    SEAL_FLATTENER_STATES.MovedFlattenersUpAndToClearance :                // Move flatteners to up state
                                                                    IF enable AND semiAutoModeSelected OR (autoModeSelected AND (_amMoveInToBagHolding OR _amMoveIn)) THEN
                                                                        state := SEAL_FLATTENER_STATES.MoveFlattenersIn;
                                                                        //ClearCommands();
                                                                    END_IF
                                        
                                                                    
    SEAL_FLATTENER_STATES.MoveFlattenersIn :                        // Move flatteners up and in
                                                                    //sealFlattenersHorizontalAxisMotor.NextSequence();    
                                                                    sealFlattenersHorizontalAxisMotor.MoveToPosition(position := inSetpoint, 
                                                                                                                        acceleration := horizontalAxisAccel,
                                                                                                                        deceleration := horizontalAxisDecel,
                                                                                                                        velocity := moveInSpeed);                                                    
                                                                    state := SEAL_FLATTENER_STATES.MovingFlattenersIn;
                                                                    
                                                                    
    SEAL_FLATTENER_STATES.MovingFlattenersIn :                        // If we did that command well move on 
                                                                        delay.IN := TRUE;
                                                                        IF delay.Q THEN
																			IF sealFlattenersHorizontalAxisMotor.CommandAcknowledged AND sealFlattenersHorizontalAxisMotor.InPosition THEN
																				state := SEAL_FLATTENER_STATES.MovedFlattenersIn;
                                                                           		delay.IN := FALSE;    
																			END_IF
                                                                        END_IF 
                                                                    
    SEAL_FLATTENER_STATES.MovedFlattenersIn :                        // Now that we're up and in move to down and 4 corners/bag holding
                                                                    IF enable AND semiAutoModeSelected OR (autoModeSelected AND _amMoveInToBagHolding) THEN
                                                                        state := SEAL_FLATTENER_STATES.MoveFlattenersDown;
                                                                        ClearCommands();
                                                                    END_IF    
    
    SEAL_FLATTENER_STATES.MoveFlattenersDown :            // Do moves for down and bag holding
                                                                        
                                                                        sealFlattenersVerticalAxis.Extend();
                                                                                                                                                                                
                                                                        state := SEAL_FLATTENER_STATES.MovingFlattenersDown;
                                                                        
    SEAL_FLATTENER_STATES.MovingFlattenersDown :            
                                                                        //IF sealFlattenersVerticalAxis.CommandAcknowledged AND sealFlattenersVerticalAxis.InPosition THEN
                                                                       	fingersDownDelay.IN := TRUE;
																	  	IF fingersDownDelay.Q THEN
																			state := SEAL_FLATTENER_STATES.MovedFlattenersDown;
																			fingersDownDelay.IN := FALSE;
																		END_IF 
																		
                                                                        //END_IF 
                                                                        
    SEAL_FLATTENER_STATES.MovedFlattenersDown :            state := SEAL_FLATTENER_STATES.MoveFlattenersToBagHolding;
                                                                    
                                                                    
    SEAL_FLATTENER_STATES.MoveFlattenersToBagHolding :            // Do moves for down and bag holding
                                                                        //sealFlattenersHorizontalAxisMotor.NextSequence();    
                                                                        sealFlattenersHorizontalAxisMotor.MoveToPositionTorque(position := bagHoldingSetpoint, 
                                                                                                                        acceleration := horizontalAxisAccel,
                                                                                                                        deceleration := horizontalAxisDecel,
                                                                                                                        velocity := moveBagHoldingSpeed,
																														current := bagHoldingCurrentMSF);                                                
                                                                        state := SEAL_FLATTENER_STATES.MovingFlattenersToBagHolding;
                                                                        
    SEAL_FLATTENER_STATES.MovingFlattenersToBagHolding :            delay.IN := TRUE;
                                                                        IF delay.Q THEN
																			IF sealFlattenersHorizontalAxisMotor.CommandAcknowledged THEN
																				state := SEAL_FLATTENER_STATES.MovedFlattenersToBagHolding;
                                                                            	delay.IN := FALSE; 
																			END_IF   
                                                                        END_IF 
                                                                        
    SEAL_FLATTENER_STATES.MovedFlattenersToBagHolding :            state := SEAL_FLATTENER_STATES.Idle;
																		HMIData.motorizedSealFlattenerCycles.Increment();
                                                                        Globals.motorizedSealFlattenersCount := Globals.motorizedSealFlattenersCount +1;
                                                                        Globals.sealFlattenerFingersCount := Globals.sealFlattenerFingersCount +1;
    SEAL_FLATTENER_STATES.Ready :
    SEAL_FLATTENER_STATES.Fault :
END_CASE

METHOD PRIVATE ClearCommands
VAR_INPUT
END_VAR
// Clear all commands from auto mode
_amMoveOut := FALSE;
_amMoveClearance := FALSE;
_amMoveInToBagHolding := FALSE;
_amMoveIn := FALSE;
END_METHOD

METHOD AutoMoveOut
VAR_INPUT
END_VAR
_amMoveOut := TRUE;
END_METHOD

PROPERTY Mode : DEVICE_MODES
SET
_mode := Mode;
END_SET
GET
Mode := _mode;
END_GET
END_PROPERTY

PROPERTY Ready : BOOL
GET
Ready := _ready;
END_GET
SET
_ready := Ready;
END_SET
END_PROPERTY

METHOD AutoMoveToClearance
VAR_INPUT
END_VAR
_amMoveClearance := TRUE;
END_METHOD

METHOD AutoMoveToBagHolding
VAR_INPUT
END_VAR
_amMoveInToBagHolding := TRUE;
END_METHOD

METHOD AutoMoveIn : BOOL
VAR_INPUT
END_VAR
_amMoveIn := TRUE;
END_METHOD

END_FUNCTION_BLOCK

// Device/Application/FBs/Cylinders/ICylinder
INTERFACE ICylinder

METHOD Extend
VAR_INPUT
END_VAR
END_METHOD

METHOD Execute
VAR_INPUT
END_VAR
END_METHOD

METHOD Retract
VAR_INPUT
END_VAR
END_METHOD

END_INTERFACE

// Device/Application/FBs/Motors/Festo/FB_FestoMotor
FUNCTION_BLOCK FB_FestoMotor IMPLEMENTS IPositionableMotor, IStoredProgramMotor
VAR_INPUT
    deviceType : FML.E_FML_DEVICE_TYPE;                            //Must define drive type
    isFPCActive : BOOL;    
    ptrReadFHPPRegister : POINTER TO WORD;
    ptrReadFPCRegister : POINTER TO WORD;
    ptrWriteFHPPRegister : POINTER TO WORD;
    ptrWriteFPCRegister : POINTER TO WORD;                                        //Toggle if FPC(Festo Parameter Chanel) is active or not
END_VAR
VAR_IN_OUT
    //modbusReadRegisters :  ARRAY[0..7] OF WORD;        //Inputs from drive
    //modbusWriteRegisters : ARRAY[0..7] OF WORD;    //Outputs to write to drive

END_VAR
VAR_OUTPUT
END_VAR
VAR
    //Required datatypes for the Festo motor blocks
    FHPP_IN     :ARRAY[0..7] OF BYTE;
    FHPP_OUT     :ARRAY[0..7] OF BYTE;
    FPC_IN         :ARRAY[0..7] OF BYTE;
    FPC_OUT     :ARRAY[0..7] OF BYTE;
    ReadAxis            :FML.FML_Read;
    DATA_REF_Axis         :FML.DT_FML_REF;
    CRTL_Axis            :FML.FHPP_CTRL;
    PNU_Axis            :FML.FPC_PNU;
    MULTI_Axis            :FML.FPC_MULTI;    
    DIRMP_Axis            :FML.FPC_DIRMP;
    DIAG_Axis            :FML.FPC_DIAG;
    DIAG_BUFF_Axis        :FML.FPC_DIAG_BUFFER;
    DATA_OBJECT_Axis    :FML.FPC_DATA_OBJECT;
    FILE_Axis            :FML.FPC_FILE;
    FILE_ARRAY_Axis        :FML.FPC_FILE_ARRAY;
    WriteAxis            :FML.FML_Write;

    //Regular variables
    ptrModbusMemory : POINTER TO ARRAY[0..7] OF BYTE; 
    commandSuccessful : BOOL;    //Modbus Command was successful
    homeRequiredIndication : BOOL; //Home required indication
    homingActive : BOOL;            //Homing active
    removeStartCommandTimer : Standard.TON := (PT := T#100MS);
    startAckONS : Standard.R_TRIG;
    _sendStart : BOOL;
END_VAR
VAR_STAT    
    //Make these static to share amongst all instances of the Festo motors
    ARY_DATA_FILE        :ARRAY[0..25000] OF BYTE;
    MultiParam             :ARRAY [0..7] OF DT_FML_PRM_DESCRIPTION :=[
                                            (PNU:=404, SUBINDEX:=1, ACCESS:=0, VALUE:=0, LENGTH:=0),
                                            (PNU:=404, SUBINDEX:=1, ACCESS:=1, VALUE:=100, LENGTH:=4),
                                            (PNU:=404, SUBINDEX:=1, ACCESS:=0, VALUE:=0, LENGTH:=0),
                                            (PNU:=404, SUBINDEX:=2, ACCESS:=0, VALUE:=0, LENGTH:=0),
                                            (PNU:=404, SUBINDEX:=2, ACCESS:=1, VALUE:=200, LENGTH:=4),
                                            (PNU:=404, SUBINDEX:=2, ACCESS:=0, VALUE:=0, LENGTH:=0),
                                            (PNU:=404, SUBINDEX:=1, ACCESS:=1, VALUE:=111, LENGTH:=4),
                                            (PNU:=404, SUBINDEX:=1, ACCESS:=0, VALUE:=0, LENGTH:=0)];
                                            
END_VAR

METHOD ExecuteStoredProgram
VAR_INPUT
    (*Program number to execute*)
    programNumber    : INT;
END_VAR
InitDrive();
IF InPosition AND CRTL_Axis.ActualRecordNo = programNumber THEN
    commandSuccessful := TRUE;
ELSE
    CRTL_Axis.RecordNo := programNumber;
    _sendStart := TRUE;
END_IF
END_METHOD

PROPERTY Homing : BOOL
GET
Homing := homingActive;
END_GET
END_PROPERTY

PROPERTY HomeRequired : BOOL
GET
HomeRequired := homeRequiredIndication;
END_GET
SET
homeRequiredIndication := HomeRequired;
END_SET
END_PROPERTY

{attribute 'monitoring' := 'variable'}
PROPERTY CurrentPosition : REAL
GET
{warning: 'TODO: Find out actual conversion factor'}    
CurrentPosition := (DINT_TO_REAL(CRTL_Axis.ActualPosition)/100);
END_GET
END_PROPERTY

METHOD Execute
VAR_INPUT
END_VAR


//Check to make sure we have a valid reference.  Disable complier warning since we're doing the check
//{warning disable C0371}
(*
IF NOT __ISVALIDREF(ptrReadFHPPRegister) 
    OR NOT __ISVALIDREF(ptrReadFPCRegister) 
    OR NOT __ISVALIDREF(ptrWriteFHPPRegister)
    OR NOT __ISVALIDREF(ptrWriteFPCRegister)
THEN
     RETURN;
END_IF
*)



//Convert array of bytes to array of words. Playin' with pointers!
ptrModbusMemory := ptrReadFHPPRegister;
FHPP_IN := ptrModbusMemory^; 
ptrModbusMemory := ptrReadFPCRegister;
FPC_IN := ptrModbusMemory^;
ptrModbusMemory := ptrWriteFHPPRegister;
ptrModbusMemory^ := FHPP_OUT; 
ptrModbusMemory := ptrWriteFPCRegister;
ptrModbusMemory^ := FPC_OUT;

// Function block calls for axis
ReadAxis(
    FML_REF            := DATA_REF_Axis,
    Modbus            := FALSE,
    HighByteFirst    := TRUE,
    DeviceType        := deviceType,
    FPC_active        := isFPCActive,
    
    FHPP_Source        := FHPP_IN,
    FPC_Source        := FPC_IN);    
CRTL_Axis(
    FML_REF            := DATA_REF_Axis);    
PNU_Axis(
    FML_REF            := DATA_REF_Axis);
MULTI_Axis(
    FML_REF            := DATA_REF_Axis,
    SizeOfParam        := SIZEOF(MultiParam),
    AdrOfParam        := ADR(MultiParam));
DIRMP_Axis(
    FML_REF            := DATA_REF_Axis);    
DIAG_Axis(
    FML_REF            := DATA_REF_Axis);
DIAG_BUFF_Axis(
    FML_REF            := DATA_REF_Axis);
DATA_OBJECT_Axis(
    FML_REF            := DATA_REF_Axis);
FILE_Axis(
    FML_REF            := DATA_REF_Axis);
FILE_ARRAY_Axis(
    FML_REF            := DATA_REF_Axis,
    SizeOfFileArray    := SIZEOF(ARY_DATA_FILE),
    AdrOfFileArray    := ADR(ARY_DATA_FILE));    
WriteAxis(
    FML_REF            := DATA_REF_Axis,
    FHPP_Target        => FHPP_OUT,
    FPC_Target        => FPC_OUT);
{warning 'TODO: Remove this hack to clear start command if error occurs'}
removeStartCommandTimer(IN := CRTL_Axis.StartTask OR CRTL_Axis.AckStart);
//removeStartCommandTimer(IN := CRTL_Axis.AckStart);
startAckONS(CLK := CRTL_Axis.AckStart);    
//IF removeStartCommandTimer.Q THEN
IF _sendStart AND NOT CRTL_Axis.AckStart THEN
    CRTL_Axis.StartTask := TRUE;
    _sendStart := FALSE;
END_IF

IF startAckONS.Q OR removeStartCommandTimer.Q THEN
    CRTL_Axis.StartTask := FALSE;
    commandSuccessful := TRUE;
END_IF
//Set Home required indication
homeRequiredIndication S= NOT CRTL_Axis.HomingValid;
//commandSuccessful S= CRTL_Axis.AckStart;
//{warning restore C0371}
END_METHOD

{attribute 'monitoring' := 'variable'}
PROPERTY CommandAcknowledged : BOOL
GET
CommandAcknowledged := commandSuccessful;
END_GET
END_PROPERTY

METHOD Stop
commandSuccessful := FALSE;
CRTL_Axis.EnableDrive := TRUE;
CRTL_Axis.Halt := TRUE;
CRTL_Axis.Stop := FALSE;
END_METHOD

{attribute 'monitoring' := 'variable'}
PROPERTY ActiveStoredProgramNumber : INT
GET
ActiveStoredProgramNumber := CRTL_Axis.ActualRecordNo;
END_GET
END_PROPERTY

METHOD PRIVATE InitDrive
VAR_INPUT
END_VAR
//Initialize the drive to prepare for a move
CRTL_Axis.EnableDrive := TRUE;
CRTL_Axis.Halt := TRUE;
CRTL_Axis.Stop := TRUE;    
//CRTL_Axis.StartTask := FALSE;
commandSuccessful := FALSE;
END_METHOD

PROPERTY Moving : BOOL
GET
Moving := CRTL_Axis.DriveIsMoving;
END_GET
END_PROPERTY

{warning 'add method implementation '}
METHOD MoveDistance
VAR_INPUT
    (*Distance to move in inches*)
    distance    : REAL;
    (*Acceleration in RPM/sec*)
    acceleration    : INT;
    (*Deceleration in RPM/sec*)
    deceleration    : INT;
    (*Velocity in .25RPM*)
    velocity    : INT;
END_VAR
END_METHOD

{attribute 'monitoring' := 'variable'}
PROPERTY InPosition : BOOL
GET
InPosition := CRTL_Axis.MC;
END_GET
END_PROPERTY

{warning 'add method implementation '}
METHOD MoveToPosition
VAR_INPUT
    (*Position to move to in inches*)
    position    : REAL;
    (*Acceleration in RPM/sec*)
    acceleration    : INT;
    (*Deceleration in RPM/sec*)
    deceleration    : INT;
    (*Velocity in .25RPM*)
    velocity    : INT;
END_VAR
END_METHOD

METHOD HomeNow
CRTL_Axis.StartHoming := TRUE;
END_METHOD

END_FUNCTION_BLOCK

// Device/Application/FBs/Motors/IPositionableMotor
INTERFACE IPositionableMotor

PROPERTY Homing : BOOL
GET
END_GET
END_PROPERTY

PROPERTY Moving : BOOL        //Motor is Moving
GET
END_GET
END_PROPERTY

PROPERTY InPosition : BOOL        //Motor is in position
GET
END_GET
END_PROPERTY

PROPERTY CurrentPosition : REAL        //Current motor position in Inches
GET
END_GET
END_PROPERTY

METHOD Stop
VAR_INPUT
END_VAR
END_METHOD

PROPERTY CommandAcknowledged : BOOL        //Command acked from drive
GET
END_GET
END_PROPERTY

METHOD HomeNow
VAR_INPUT
END_VAR
END_METHOD

METHOD MoveToPosition
VAR_INPUT
    position : REAL;        //Position to move to in inches
    acceleration : INT;        //Acceleration in RPM/sec
    deceleration : INT;        //Deceleration in RPM/sec
    velocity : INT;            //Velocity in .25RPM
END_VAR
END_METHOD

PROPERTY HomeRequired : BOOL
GET
END_GET
SET
END_SET
END_PROPERTY

METHOD MoveDistance
VAR_INPUT
    distance : REAL;        //Distance to move in inches
    acceleration : INT;        //Acceleration in RPM/sec
    deceleration : INT;        //Deceleration in RPM/sec
    velocity : INT;            //Velocity in .25RPM
END_VAR
END_METHOD

END_INTERFACE

// Device/Application/FBs/Motors/IStoredProgramMotor
INTERFACE IStoredProgramMotor

PROPERTY ActiveStoredProgramNumber : INT
GET
END_GET
END_PROPERTY

METHOD ExecuteStoredProgram
VAR_INPUT
    programNumber : INT;        //Program number to execute
END_VAR
END_METHOD

END_INTERFACE

// Device/Application/FBs/Fault/FB_ONS
FUNCTION_BLOCK FB_ONS
VAR_INPUT
	CLK : BOOL;
END_VAR
VAR_OUTPUT
	OSR : BOOL;
	OSF : BOOL;
END_VAR
VAR
	CLK_OSR : R_TRIG;
	CLK_OSF : F_TRIG;
END_VAR

CLK_OSR(CLK := CLK, Q=> OSR);
CLK_OSF(CLK := CLK, Q=> OSF);

END_FUNCTION_BLOCK

// Device/Application/FBs/Motors/Applied Motion/FB_AppliedMotionStepServoEIPBaseQX
FUNCTION_BLOCK FB_AppliedMotionStepServoEIPBaseQX IMPLEMENTS IPositionableMotor, IStoredProgramMotor
VAR_INPUT
    ptrEIPInputs : POINTER TO ARRAY[0..13] OF  DINT;
    ptrEIPOutputs : POINTER TO ARRAY[0..15] OF DINT;
    faultHandler : REFERENCE TO FB_FaultHandler;
	commFail : BOOL;
    stepsPerInchSetpoint : INT;             //Steps per inch setpoint
    reversePolarity : BOOL;                 //0 = Normal, 1 = reversed polarity for display
    jogAccelSetpoint : INT;        //Point-to-Point Acceleration (AC) Setpoint
    jogDecelSetpoint : INT;        //Point-to-Point Deceleration (DE) Setpoint
    jogVelocitySetpoint : INT;                //Velocity (VE) Setpoint
    pointToPointAccelSetpoint : INT;        //Point-to-Point Acceleration (AC) Setpoint
    pointToPointDecelSetpoint : INT;        //Point-to-Point Deceleration (DE) Setpoint
    velocitySetpoint : INT;                //Velocity (VE) Setpoint
	defaultCurrentSetpoint : DINT;
	sclCommand : DINT;						// SCL Command from 
	parameter1 : DINT;						// Data/SCL parameter 1
	parameter2 : DINT;						// Data/SCL parameter 2
    distanceSetpointInches : REAL;        //Distance setpoint in inches Setpoint
    moveDistanceManualPB : BOOL;            //Move distance pushbutton
    movePositionManualPB : BOOL;            //Move position pushbutton
	isHomable : BOOL;
END_VAR
VAR_IN_OUT
    //slave : IoDrvModbusTCP.ModbusTCPSlave;                    //Slave ModbusTCP Object
END_VAR
VAR
    absolutePositionSteps : DINT; //Immediate Absolute Position in steps
    distanceToMoveInSteps : DINT;        //Distance Setpoint to Drive
    stepServoStatusRaw : INT; //Raw step servo status over modbus
	stepServoAlarmCodeRaw : INT; // Ras Step Servo alarm code word
	currentLimit : DINT;
    commands : FB_StepServoCommands();
    commandSuccessful : BOOL;    //Modbus Command was successful
    commandSuccessfulONS : R_TRIG;    //Modbus Command was successful
    commandSentONS : R_TRIG;    //Modbus Command was successful
    homeRequiredIndication : BOOL; //Home required indication.
    driveInputs : ARRAY[0..13] OF DINT;        // Inputs from drive over EIP
    driveOutputs : ARRAY[0..15] OF DINT;    // Outputs to drive over EIP
    interfaceToPass : IFault;
    faultListRegisterSuccess : BOOL;        // Registering in fault list successful
    _faulted : BOOL;                    // Motor Faulted
	_reset : BOOL;			//Reset Motor
	_homeNow : BOOL;
	homingOSF : F_TRIG;
	
	IECReferenceGood : BOOL;
END_VAR
VAR_OUTPUT
    absolutePositonInches : REAL; //Immediate Absolute Positon in inches
    velocity : INT;    //Velocity (VE) Input from Drive
    status : StepServoStatusFB; //Status of servo
	alarms : FB_StepServoAlarms; // Alarms from Drive
    QSegmentRunning : INT; //Current Q program running from Drive
	faults : StepServoFaultsType;
END_VAR


IF NOT faultListRegisterSuccess THEN
    faultListRegisterSuccess := RegisterWithFaultHandler();
END_IF

METHOD Execute
VAR_INPUT
END_VAR
//    Function Block: AppliedMotionStepServo
//    Description: This block provides an abstraction for a Ethernet I/P Applied Motion Step Servo
//    Created by: Ben Hess
//    Created Date: May 11th, 2018

// Use pointers for EIP memory register locations
driveInputs := ptrEIPInputs^;

ptrEIPOutputs^ := driveOutputs;
alarms(alarmCode := stepServoAlarmCodeRaw, faults := faults);

IF currentLimit = 0 THEN 
	currentLimit := defaultCurrentSetpoint;
END_IF
//Map raw EIP Registers to parameters
absolutePositionSteps := driveInputs[6];
velocity := DINT_TO_INT(driveInputs[8]);
stepServoStatusRaw := DINT_TO_INT(driveInputs[0]);

driveOutputs[4] := velocitySetpoint;
driveOutputs[5] := pointToPointAccelSetpoint;
driveOutputs[6] := pointToPointDecelSetpoint;
driveOutputs[7] := distanceToMoveInSteps;
driveOutputs[8] := currentLimit;
driveOutputs[9] := sclCommand;
driveOutputs[10] := parameter1;
driveOutputs[11] := parameter2;
driveOutputs[12] := currentLimit;
driveOutputs[13] := currentLimit + 1;
driveOutputs[0] := commands.commandWord;
// Step servo command bits handler
commands();
//Convert Distance setpoint to steps.  Reverse polarity for display purposes if needed. 

absolutePositonInches := (DINT_TO_REAL(absolutePositionSteps) / INT_TO_REAL(stepsPerInchSetpoint));

//Homing required from motor - for now just if there was an initialization seen.
homeRequiredIndication S= status.initializing OR Globals.firstScan OR _faulted OR driveInputs[11].0;

homingOSF(CLK := status.homing);
IF NOT driveInputs[11].0 THEN
	homeRequiredIndication := FALSE;
END_IF

commandSentONS(CLK := commands.commandSent);

IF commandSentONS.Q THEN
	commandSuccessful := TRUE;
END_IF

commandSuccessfulONS(CLK := commandSuccessful);
IF commandSuccessfulONS.Q THEN
	//parameter1 := 0;
	//velocitySetpoint := 0;
	//pointToPointAccelSetpoint := 0;
	//pointToPointDecelSetpoint := 0;
	//distanceToMoveInSteps := 0;
END_IF


IF _reset AND (status.driveFaulted OR status.alarmPresent) THEN
	commands.alarmReset := TRUE;
	_reset := FALSE;
END_IF

IF reversePolarity THEN
    absolutePositonInches := absolutePositonInches * -1; 
END_IF

//Get Servo Status and unpack
status(statusCode := StepServoStatusRaw);

//Bit-packing for LONG types over Modbus

_faulted := status.driveFaulted OR status.alarmPresent OR commFail;

//Manual moves for motor
IF moveDistanceManualPB THEN
    MoveDistance(distance := distanceSetpointInches, acceleration := pointToPointAccelSetpoint, deceleration := pointToPointDecelSetpoint, velocity := velocitySetpoint);
    moveDistanceManualPB := FALSE;
END_IF

IF movePositionManualPB THEN
    MoveToPosition(position := distanceSetpointInches, acceleration := pointToPointAccelSetpoint, deceleration := pointToPointDecelSetpoint, velocity := velocitySetpoint);
    movePositionManualPB := FALSE;
END_IF


faults.commFail.faultTrigger := commFail AND Globals.machinePowerOK;
faults.notHomed.faultTrigger := homeRequiredIndication AND isHomable;
END_METHOD

{attribute 'monitoring' := 'variable'}
PROPERTY CommandAcknowledged : BOOL
GET
CommandAcknowledged := commandSuccessful;
END_GET
END_PROPERTY

METHOD HomeNow
commandSuccessful := FALSE;
parameter1 := 1;
pointToPointAccelSetpoint := 1000;
pointToPointDecelSetpoint := 1000;
velocitySetpoint := 2500;
distanceToMoveInSteps := 0;
commands.sendQAndExecute := TRUE;

//homeRequiredIndication := FALSE;
END_METHOD

{attribute 'monitoring' := 'variable'}
PROPERTY HomeRequired : BOOL
SET
homeRequiredIndication := HomeRequired;
END_SET
GET
HomeRequired := homeRequiredIndication;
END_GET
END_PROPERTY

{attribute 'monitoring' := 'variable'}
PROPERTY Moving : BOOL
GET
Moving := status.moving;
END_GET
END_PROPERTY

{attribute 'monitoring' := 'variable'}
PROPERTY ActiveStoredProgramNumber : INT
GET
ActiveStoredProgramNumber := QSegmentRunning;
END_GET
END_PROPERTY

{attribute 'monitoring' := 'variable'}
PROPERTY InPosition : BOOL
GET
InPosition := status.inPosition;
END_GET
END_PROPERTY

METHOD MoveDistanceTorque
VAR_INPUT
	(*Distance to move in inches*)
    distance    : REAL;
    (*Acceleration in RPM/sec*)
    acceleration    : INT;
    (*Deceleration in RPM/sec*)
    deceleration    : INT;
    (*Velocity in .25RPM*)
    velocity    : INT;
	(*Current in .01A*)
	current : DINT;
END_VAR
//This method preps the data to send to the drive and triggers the send.
//Set distance and unpack to prep data to send to motor

commandSuccessful := FALSE;

distanceToMoveInSteps := REAL_TO_DINT((distance) * stepsPerInchSetpoint);
IF reversePolarity THEN
    distanceToMoveInSteps := distanceToMoveInSteps * -1;
END_IF

pointToPointAccelSetpoint := acceleration;
pointToPointDecelSetpoint := deceleration;
velocitySetpoint := velocity;
currentLimit := current;

parameter1 := 2;
commands.SendQAndExecute := TRUE;
END_METHOD

(* This will be called if the machine is faulted*)
METHOD MachineFaulted
END_METHOD

{attribute 'monitoring' := 'variable'}
PROPERTY Faulted : BOOL
GET
Faulted := _faulted;
END_GET
SET
END_SET
END_PROPERTY

METHOD MoveToPosition
VAR_INPUT
    (*Position to move to in inches*)
    position    : REAL;
    (*Acceleration in RPM/sec*)
    acceleration    : INT;
    (*Deceleration in RPM/sec*)
    deceleration    : INT;
    (*Velocity in .25RPM*)
    velocity    : INT;
END_VAR
commandSuccessful := FALSE;

distanceToMoveInSteps := REAL_TO_DINT((position) * stepsPerInchSetpoint);
IF reversePolarity THEN
    distanceToMoveInSteps := distanceToMoveInSteps * -1;    
END_IF

pointToPointAccelSetpoint := acceleration;
pointToPointDecelSetpoint := deceleration;
velocitySetpoint := velocity;
currentLimit := defaultCurrentSetpoint;

commands.feedToPosition := TRUE;
END_METHOD

METHOD MoveToPositionTorque
VAR_INPUT
	(*Position to move to in inches*)
    position    : REAL;
    (*Acceleration in RPM/sec*)
    acceleration    : INT;
    (*Deceleration in RPM/sec*)
    deceleration    : INT;
    (*Velocity in .25RPM*)
    velocity    : INT;
	(*Current in .01A*)
	current : DINT;
END_VAR
commandSuccessful := FALSE;

distanceToMoveInSteps := REAL_TO_DINT((position) * stepsPerInchSetpoint);
IF reversePolarity THEN
    distanceToMoveInSteps := distanceToMoveInSteps * -1;    
END_IF

pointToPointAccelSetpoint := acceleration;
pointToPointDecelSetpoint := deceleration;
velocitySetpoint := velocity;
currentLimit := current;

commands.feedToPosition := TRUE;
THIS^.Execute();
END_METHOD

//{warning 'add method implementation '}
METHOD Stop
commandSuccessful := FALSE;
commands.StopNormal := TRUE;
END_METHOD

METHOD MoveDistance
VAR_INPUT
    (*Distance to move in inches*)
    distance    : REAL;
    (*Acceleration in RPM/sec*)
    acceleration    : INT;
    (*Deceleration in RPM/sec*)
    deceleration    : INT;
    (*Velocity in .25RPM*)
    velocity    : INT;
END_VAR
//This method preps the data to send to the drive and triggers the send.
//Set distance and unpack to prep data to send to motor

commandSuccessful := FALSE;

distanceToMoveInSteps := REAL_TO_DINT((distance) * stepsPerInchSetpoint);
IF reversePolarity THEN
    distanceToMoveInSteps := distanceToMoveInSteps * -1;
END_IF

pointToPointAccelSetpoint := acceleration;
pointToPointDecelSetpoint := deceleration;
velocitySetpoint := velocity;
currentLimit := defaultCurrentSetpoint;

commands.feedToLength := TRUE;
END_METHOD

{attribute 'monitoring' := 'variable'}
PROPERTY CurrentPosition : REAL  //Current motor position in Inches
GET
CurrentPosition := absolutePositonInches;
END_GET
END_PROPERTY

{attribute 'monitoring' := 'variable'}
PROPERTY Homing : BOOL
GET
Homing := status.homing;
END_GET
END_PROPERTY

METHOD Reset : BOOL
VAR_INPUT
END_VAR
IF Faulted THEN
	_reset := TRUE;
	commands.AlarmReset := TRUE;
END_IF
commands.Enable := TRUE;
END_METHOD

METHOD RegisterWithFaultHandler : BOOL
// If faulthandler hasn't been initialized yet then do nothing.

(*
IF NOT __ISVALIDREF(faultHandler) THEN
     RETURN;
END_IF

interfaceToPass := THIS^;
faultHandler.registerFaultSource(interfaceToPass);
RegisterWithFaultHandler := TRUE;
*)
END_METHOD

METHOD ExecuteStoredProgram
VAR_INPUT
    (*Program number to execute*)
    programNumber    : INT;
END_VAR
parameter1 := programNumber;
commands.SendQAndExecute := TRUE;
END_METHOD

END_FUNCTION_BLOCK

// Device/Application/FBs/FB_FaultHandler
FUNCTION_BLOCK FB_FaultHandler
VAR_INPUT
END_VAR
VAR_OUTPUT
END_VAR
VAR
    faultSourceList : ARRAY[0..100] OF IFault;
    sourcesInList : INT;
END_VAR

METHOD registerFaultSource
VAR_INPUT
     faultSource : REFERENCE TO IFault;
END_VAR
faultSourceList[sourcesInList]:= faultSource;
sourcesInList:= sourcesInList + 1;
END_METHOD

END_FUNCTION_BLOCK

// Device/Application/ObjectHandling/IFault
INTERFACE IFault EXTENDS IAllObjects

METHOD Trigger
VAR_INPUT
END_VAR
END_METHOD

METHOD Ack
VAR_INPUT
END_VAR
END_METHOD

END_INTERFACE

// Device/Application/ObjectHandling/IAllObjects
INTERFACE IAllObjects EXTENDS __System.IQueryInterface

PROPERTY InstanceName : STRING
GET
END_GET
END_PROPERTY

END_INTERFACE

// Device/Application/FBs/Motors/Applied Motion/DataHandlers/FB_StepServoCommands
{analysis -166, -35, -36, -38, -148}
FUNCTION_BLOCK FB_StepServoCommands
VAR_INPUT
       
END_VAR
VAR_OUTPUT
    commandWord : DINT;
	commandSent : BOOL;
END_VAR
VAR
	_idleState : BOOL; // Idle State (Send this between repeated commands)
    _enable : BOOL; // Enable
    _disable : BOOL; // Disable
    _feedToLength : BOOL; // Start Move - FL
    _feedToPosition : BOOL; // Start Move - FP
    _feedToSensor : BOOL; // Start Move - FS (sensor)
    _feedToDoubleSensor : BOOL; // Start Move - FD (double sensor)
    _feedToSensorSafety : BOOL; // Start Move - FY (sensor w/ safety distance)
    _feedToSensorMask : BOOL; // Start Move - FM (sensor w/ mask distance)
    _feedAndSetOutput : BOOL; // Start Move - FO (set output)
    _feedSpeedChange : BOOL; // Start Move - FC
    _seekHome : BOOL; // Start Move - SH
    _findHome : BOOL; // Start Move - FH
    _followEncoder : BOOL; // Start Move - FE
    _stopAndKillCrash : BOOL; // Stop/Kill - AM
    _stopAndKillNormal : BOOL; // Stop/Kill - DE
    _startJog : BOOL; // Start Jogging
    _updateJogSpeed : BOOL; // Update Jog Speed
    _sendHostCommand : BOOL; // Send Host Command
    _sendQAndExecute : BOOL; // Q Load & Execute (QX)
    _alarmReset : BOOL; // Alarm Reset - AR 
	clearCommandWordTimer : TON := (PT := REAL_TO_TIME(INT_TO_REAL(Globals.AMP_MOTOR_RPI) * 1.5));
	clearCommandWordTimer2 : TON := (PT := REAL_TO_TIME(INT_TO_REAL(Globals.AMP_MOTOR_RPI) * 1.5));
END_VAR

{analysis -166, -35, -36, -148}
//    Fucntion Block: FB_StepServoCommands
//    Description: This packs the step servo command bits into the register send over EIP
//    Created by: Ben Hess
//    Created Date: May 11th, 2018

// Set the proper output bit
commandWord.0 := _idleState;
commandWord.1 := _enable;
commandWord.2 := _disable;
commandWord.3 := _feedToLength;
commandWord.4 := _feedToPosition;
commandWord.5 := _feedToSensor;
commandWord.6 := _feedToDoubleSensor;
commandWord.7 := _feedToSensorSafety;
commandWord.8 := _feedToSensorMask;
commandWord.9 := _feedAndSetOutput;
commandWord.10 := _feedSpeedChange;
commandWord.11 := _seekHome;
commandWord.12 := _findHome;
commandWord.13 := _followEncoder;
commandWord.14 := _stopAndKillCrash;
commandWord.15 := _stopAndKillNormal;
commandWord.16 := _startJog;
commandWord.17 := _updateJogSpeed;
commandWord.18 := _sendHostCommand;
commandWord.19 := _sendQAndExecute;
commandWord.20 := _alarmReset;


// CLear the command bits after 1.3x motor RPI
clearCommandWordTimer(IN := commandWord <> 0);
clearCommandWordTimer2();
IF clearCommandWordTimer.Q THEN
	THIS^.Clear();
	clearCommandWordTimer2.IN := TRUE;
END_IF

IF clearCommandWordTimer2.Q THEN
		commandSent := TRUE;
		clearCommandWordTimer2.IN := FALSE;
END_IF

PROPERTY Enable : BOOL
SET
commandSent := FALSE;
_enable := Enable;
END_SET
GET
Enable := _enable;
END_GET
END_PROPERTY

PROPERTY AlarmReset : BOOL
GET
AlarmReset := _alarmReset;
END_GET
SET
commandSent := FALSE;
_alarmReset := AlarmReset;
END_SET
END_PROPERTY

PROPERTY SendHostCommand : BOOL
GET
SendHostCommand := _sendHostCommand;
END_GET
SET
commandSent := FALSE;
_sendHostCommand := SendHostCommand;
END_SET
END_PROPERTY

PROPERTY FeedToLength : BOOL
SET
commandSent := FALSE;
_feedToLength := FeedToLength;
END_SET
GET
FeedToLength := _feedToLength;
END_GET
END_PROPERTY

METHOD Clear
VAR_INPUT
END_VAR
_idleState := FALSE;
_enable := FALSE;
_disable := FALSE;
_feedToLength := FALSE;
_feedToPosition := FALSE;
_feedToSensor := FALSE;
_feedToDoubleSensor := FALSE;
_feedToSensorSafety := FALSE;
_feedToSensorMask := FALSE;
_feedAndSetOutput := FALSE;
_feedSpeedChange := FALSE;
_seekHome := FALSE;
_findHome := FALSE;
_followEncoder := FALSE;
_stopAndKillCrash := FALSE;
_stopAndKillNormal := FALSE;
_startJog := FALSE;
_updateJogSpeed := FALSE;
_sendHostCommand := FALSE;
_sendQAndExecute := FALSE;
_alarmReset := FALSE;
END_METHOD

PROPERTY StopNormal : BOOL
SET
commandSent := FALSE;
_stopAndKillNormal := StopNormal;
END_SET
GET
StopNormal := _stopAndKillNormal;
END_GET
END_PROPERTY

PROPERTY IdleState : BOOL
GET
IdleState := _idleState;
END_GET
SET
commandSent := FALSE;
_idleState := IdleState;
END_SET
END_PROPERTY

PROPERTY Disable : BOOL
GET
Disable := _disable;
END_GET
SET
commandSent := FALSE;
_disable := Disable;
END_SET
END_PROPERTY

PROPERTY StopCrash : BOOL
SET
commandSent := FALSE;
_stopAndKillCrash := StopCrash;
END_SET
GET
StopCrash := _stopAndKillCrash;
END_GET
END_PROPERTY

PROPERTY SendQAndExecute : BOOL
GET
SendQAndExecute := _sendQAndExecute;
END_GET
SET
commandSent := FALSE;
_sendQAndExecute := SendQAndExecute;
END_SET
END_PROPERTY

PROPERTY FeedToPosition : BOOL
SET
commandSent := FALSE;
_feedToPosition := FeedToPosition;
END_SET
GET
FeedToPosition := _feedToPosition;
END_GET
END_PROPERTY

END_FUNCTION_BLOCK

// Device/Application/FBs/Motors/Applied Motion/DataHandlers/StepServoStatusFB
FUNCTION_BLOCK StepServoStatusFB
VAR_INPUT
    statusCode : INT;
END_VAR
VAR_OUTPUT
    motorEnabled : BOOL;        //Motor Enabled (Motor Disabled if this bit = 0)
    sampling : BOOL;      //Sampling (for Quick Tuner)
    driveFaulted : BOOL;      //Drive Fault (check Alarm Code)
    inPosition : BOOL;      //In Position (motor is in position)
    moving : BOOL;      //Moving (motor is moving)
    jogging    : BOOL;      //Jogging (currently in jog mode)
    stopping : BOOL;      //Stopping (in the process of stopping from a stop command)
    waitingForInput : BOOL;      //Waiting (for an input; executing a WI command)
    saving : BOOL;      //Saving (parameter data is being saved)
    alarmPresent : BOOL;      //Alarm present (check Alarm Code)
    homing : BOOL;      //Homing (executing an SH command)
    waitingForTime : BOOL;      //Waiting (for time; executing a WD or WT command)
    wizardRunning : BOOL;      //Wizard running (Timing Wizard is running)
    checkingEncoder    : BOOL;      //Checking encoder (Timing Wizard is running)
    Q_ProgramRunning : BOOL;      //Q Program is running
    initializing : BOOL;      //Initializing (happens at power up) ; Servo Ready (for SV200 drives only)
END_VAR
VAR
END_VAR

//    Fucntion Block: StepServoStatus
//    Description: This unpacks the step servo status bits from the status word received over modbus
//    Created by: Ben Hess
//    Created Date: January 26th, 2018

motorEnabled := statusCode.0;
sampling := statusCode.1;
driveFaulted := statusCode.2;
inPosition := statusCode.3;
moving := statusCode.4;
jogging := statusCode.5;
stopping := statusCode.6;
waitingForInput    := statusCode.7;
saving := statusCode.8;
alarmPresent := statusCode.9;
homing := statusCode.10;
waitingForTime := statusCode.11;
wizardRunning := statusCode.12;
checkingEncoder := statusCode.13;
Q_ProgramRunning := statusCode.14;
initializing := statusCode.15;

END_FUNCTION_BLOCK

// Device/Application/FBs/Motors/Applied Motion/DataHandlers/FB_StepServoAlarms
FUNCTION_BLOCK FB_StepServoAlarms
VAR_INPUT
    alarmCode : INT;
END_VAR
VAR_OUTPUT
    positionLimit : BOOL;        // FAULT - Motor exceeded position limit - following error
    CCWLimit : BOOL;      // WARNING - Motor is at CCW Limit
    CWLimit : BOOL;      // WARNING - Motor is at CW Limit
    overTemp : BOOL;      // FAULT - Motor Over Temperature Limit
    internalVoltage : BOOL;      // FAULT - Internal Voltage Fault
    overVoltage    : BOOL;      // FAULT - Overvoltage Fault
    underVoltage : BOOL;      // WARNING - Undervoltage Warning
    overCurrent : BOOL;      // FAULT - Motor Overcurrent
    openMotorWinding : BOOL;      // FAULT - Motor Detected Open Winding
    badEncoder : BOOL;      // FAULT - Motor Encoder Failure
    commError : BOOL;      // WARNING - Communications Error
    badFlash : BOOL;      // WARNING - Bad Flash
    noMove : BOOL;      // WARNING - No Move
    currentFoldback    : BOOL;      // WARNING - Current Foldback
    blankQSegment : BOOL;      // WARNING - Blank Q Segment
    NVMemoryDoubleError : BOOL;      // WARNING - NV Memory Double Error
END_VAR
VAR
END_VAR
VAR_IN_OUT
	faults : StepServoFaultsType;
END_VAR

//    Fucntion Block: FB_StepServoAlarms
//    Description: This unpacks the step servo alarm bits from the alarm word received over EIP
//    Created by: Ben Hess
//    Created Date: September 5th, 2018

positionLimit := alarmCode.0;
CCWLimit := alarmCode.1;
CWLimit := alarmCode.2;
overTemp := alarmCode.3;
internalVoltage := alarmCode.4;
overVoltage := alarmCode.5;
underVoltage := alarmCode.6;
overCurrent    := alarmCode.7;
openMotorWinding := alarmCode.8;
badEncoder := alarmCode.9;
commError := alarmCode.10;
badFlash := alarmCode.11;
noMove := alarmCode.12;
currentFoldback := alarmCode.13;
blankQSegment := alarmCode.14;
NVMemoryDoubleError := alarmCode.15;

END_FUNCTION_BLOCK

// Device/Application/Programs/Faults
PROGRAM Faults
VAR
	reverseFault : FB_HMIFault;
END_VAR

reverseFault(refFault := PRG_Bagger.moabHead.bagDelivery.reverseFault);

END_PROGRAM

// Device/Application/FBs/Fault/FB_HMIFault
FUNCTION_BLOCK FINAL FB_HMIFault IMPLEMENTS IExecuteAutomatically, IAllObjects, IInitializable
VAR_INPUT
	refFault : REFERENCE TO FB_Fault;
END_VAR
VAR_OUTPUT
END_VAR
VAR
	active : REFERENCE TO BOOL;
	acknowledged : REFERENCE TO BOOL;
	ackCommand : REFERENCE TO BOOL;
	_instanceName : STRING := 'HMI Fault';
END_VAR

METHOD FB_Init : BOOL
VAR_INPUT
  bInitRetains : BOOL; // TRUE: the retain variables are initialized (reset warm / reset cold)
  bInCopyCode : BOOL;  // TRUE: the instance will be copied to the copy code afterward (online change)
END_VAR
GlobalObjects.CollectionOfAllObjects.AddObject(THIS^);
END_METHOD

METHOD FB_Reinit : BOOL
VAR_INPUT
END_VAR
THIS^.Initialize();
END_METHOD

METHOD Initialize
VAR_INPUT
END_VAR
active REF= refFault.active;
acknowledged REF= refFault.acknowledged;
ackCommand  REF= refFault.ackCommand;
_instanceName := CONCAT('HMI Fault - ', refFault.InstanceName);
END_METHOD

PROPERTY InstanceName : STRING
GET
InstanceName := _instanceName;
END_GET
END_PROPERTY

METHOD Execute
VAR 
	
END_VAR
END_METHOD

END_FUNCTION_BLOCK

// Device/Application/ObjectHandling/IExecuteAutomatically
INTERFACE IExecuteAutomatically EXTENDS IAllObjects

METHOD Execute
VAR_INPUT
END_VAR
END_METHOD

END_INTERFACE

// Device/Application/ObjectHandling/IInitializable
INTERFACE IInitializable EXTENDS IAllObjects

METHOD Initialize
VAR_INPUT
END_VAR
END_METHOD

END_INTERFACE

// Device/Application/FBs/Fault/FB_Fault
FUNCTION_BLOCK FINAL FB_Fault IMPLEMENTS IFault, ILoggable, IExecuteAutomatically
VAR_INPUT
	ackCommand : BOOL;
	faultTrigger : BOOL;
END_VAR
VAR_OUTPUT
	acknowledged : BOOL;
	active : BOOL;
END_VAR
VAR
	_active : BOOL;
	_acked : BOOL;
	_ackCommand : BOOL;
	_logger : IMachineLogger;
	ackCommandOSR : R_TRIG;
	faultTriggerONS : FB_ONS;
	activeONS : FB_ONS;
	_instanceName : STRING;
END_VAR
VAR_IN_OUT
	
END_VAR

METHOD Execute
//	Function Block: FB_Fault
//	Description: Faults should be of this FB type.  
//  An associated FaultType variable needs to be declared in the HMIData global variable list in order to be exposed via OPCUA 
//	Implementation should look as follows:
//
//  *** Instantiate the fault with constructor that contains the fault name: ***
//  VAR (*Faults*)
//		exampleFault1 : FB_Fault(name := CONCAT(_prefix,  'Example Fault 1'));
//		exampleFault2 : FB_Fault(name := CONCAT(_prefix,  'Example Fault 2'));
//  END_VAR
//
//  *** In alarm area of FB call the fault(s). refHMIFaults is passed in from above***
//  IF __ISVALIDREF(refHMIFaults) THEN
//		exampleFault1(HMIFault := refHMIFaults.exampleFault1);
//		exampleFault2(HMIFault := refHMIFaults.exampleFault2, faultTrigger := someFaultCondition);
//  END_IF
//
//	*** Either assign faultTrigger in call (as in exampleFault2 above) or set it later in logic
//	exampleFault1.faultTrigger := someFaultCondition;
//
//	Created by: Ben Hess
//	Created Date: Tuesday, May 22, 2018


{warning 'TODO: Add reference to device faulted indicaiton?'}
ackCommandOSR(CLK := _ackCommand);
faultTriggerONS(CLK := faultTrigger);
activeONS(CLK := _active);

IF faultTriggerONS.OSR THEN
	Trigger();
END_IF

IF ackCommandOSR.Q THEN
	_acked := TRUE;
	_ackCommand := FALSE;
END_IF

IF _acked AND NOT faultTrigger THEN
	_active := FALSE;
	_acked := FALSE;
END_IF

IF activeONS.OSF THEN
	GlobalObjects.CollectionOfActiveFaults.RemoveObject(THIS^);
	_logger.AddLogItem(CONCAT(InstanceName, ' Cleared'));
END_IF

// The following is for external communication to HMI etc.
IF ackCommand THEN
	Ack();
	ackCommand := FALSE;
END_IF
active := _active;
acknowledged := _acked;
END_METHOD

PROPERTY InstanceName : STRING
GET
InstanceName := _instanceName;
END_GET
END_PROPERTY

METHOD RegisterLogger
VAR_INPUT
	internalLogger : IMachineLogger;
END_VAR
_logger := internalLogger;
END_METHOD

METHOD Ack
IF _ackCommand OR _acked THEN
	RETURN;
END_IF
_acked := TRUE;
// Log the ACK.
_logger.AddLogItem(CONCAT(InstanceName,  ' Acked'));
END_METHOD

METHOD Trigger
IF _active = TRUE THEN
	RETURN;
END_IF
_active := TRUE;
GlobalObjects.CollectionOfActiveFaults.AddObject(THIS^);
IF _logger <> 0 THEN
	_logger.AddLogItem(CONCAT(InstanceName,  ' Active'));
END_IF
END_METHOD

METHOD FB_Init : BOOL
VAR_INPUT
  bInitRetains : BOOL; // TRUE: the retain variables are initialized (reset warm / reset cold)
  bInCopyCode : BOOL;  // TRUE: the instance will be copied to the copy code afterward (online change)
  name : STRING;
END_VAR
_instanceName := name;
GlobalObjects.CollectionOfAllObjects.AddObject(THIS^);
END_METHOD

END_FUNCTION_BLOCK

// Device/Application/ObjectHandling/ILoggable
INTERFACE ILoggable EXTENDS IAllObjects

METHOD RegisterLogger
VAR_INPUT
	internalLogger : IMachineLogger;
END_VAR
END_METHOD

END_INTERFACE

// Device/Application/ObjectHandling/IMachineLogger
INTERFACE IMachineLogger EXTENDS IAllObjects

METHOD AddLogItem
VAR_INPUT
	message : STRING;
END_VAR
END_METHOD

END_INTERFACE

// Device/Application/FBs/Cylinders/FB_ThreePositionCylinder
FUNCTION_BLOCK FB_ThreePositionCylinder EXTENDS FB_Cylinder IMPLEMENTS IThreePositonCylinder
VAR_INPUT
END_VAR
VAR_OUTPUT
END_VAR
VAR
END_VAR

METHOD Exhaust
extendOutput := FALSE;
retractOutput := FALSE;
END_METHOD

END_FUNCTION_BLOCK

// Device/Application/FBs/Cylinders/FB_Cylinder
FUNCTION_BLOCK FB_Cylinder IMPLEMENTS ICylinder
VAR_INPUT
    mode : DEVICE_MODES;
END_VAR
VAR_OUTPUT
    extendedStatus : BOOL;
    retractedStatus : BOOL;
    extendOutput : BOOL;
    retractOutput : BOOL;
END_VAR
VAR
END_VAR

METHOD Retract
extendOutput := FALSE;
retractOutput := TRUE;
END_METHOD

METHOD Extend
extendOutput := TRUE;
retractOutput := FALSE;
END_METHOD

METHOD Execute
//Do nothing
END_METHOD

END_FUNCTION_BLOCK

// Device/Application/FBs/Cylinders/IThreePositonCylinder
INTERFACE IThreePositonCylinder EXTENDS ICylinder

METHOD Exhaust
VAR_INPUT
END_VAR
END_METHOD

END_INTERFACE

// Device/Application/FBs/Components/PneumaticPressureBarFB_1
FUNCTION_BLOCK PneumaticPressureBarFB_1 EXTENDS BaseComponentFB
VAR_INPUT
	iPressureBarRetracted : BOOL;
	iPressureBarExtended : BOOL;
	iPressureBarNotObstructed : BOOL;
END_VAR
VAR_OUTPUT
    state : PRESSURE_BAR_STATES;     //Jaw State
	oExtendCylinder : BOOL;
	oRetractCylinder : BOOL;
	faults : PressureBarFaultsType;
END_VAR
VAR
    _amOpenJaw : BOOL;    // Auto Mode Open Jaw Command
    _amCloseJaw : BOOL;     // Auto Mode Close Jaw Command
    startCyclePB : BOOL;                //Start Cycle
    stopCyclePB : BOOL;                //Stop Cycle
    manualExtendHighPressurePB : BOOL;            //Manually Extend Cylinder High Pressure
    manualExtendLowPressurePB : BOOL;            //Manually Extend Cylinder Low Pressure
    manualRetractPB : BOOL;            //Manually Retract Cylinder
    manualExhaustPB : BOOL;            //Manually Echaust Cylinder
    timerExtendedDebounce : TON;            //Timer for extend delay
    timerExtendDwell : TON;            //Timer for extend dwell after extended
    timerRetractedDebounce : TON;        //Timer for retract delay
    timerRetractDwell : TON;        //Timer for retract dwell after extended
    timerSealDwell : TON;            //Timer for seal dwell
	timerObsSwitchFault : Standard.TON;
    extendDelaySP : INT := 50;    //Extend delay SP
    extendDwellSP : INT := 300;    //Extend dwell SP
    retractDelaySP : INT := 50;        //Retract delay SP
    retractDwellSP : INT := 750;    //Retract dwell SP
    incrementCount : R_TRIG();
    incrementSealBarCountONS : Standard.R_TRIG;
    incrementBagOpenFinersONS : Standard.R_TRIG;
	faultTimer : Standard.TON;
END_VAR
VAR_IN_OUT
	cumulativeHeadCycleCount : DINT;
END_VAR

//    Function Block: Cylinder
//    Description: This program moves a jaw cylinder back and forth
//    Created by: Ben Hess
//    Created Date: January 16th, 2017

SUPER^();

//Stop the auto cycle if button pressed or coming out of auto mode or moving the servo.
IF stopCyclePB OR NOT (_mode = DEVICE_MODES.SemiAuto) THEN 
    startCyclePB := FALSE;
END_IF

HMIData.pressureBarService.retractedFeedback := iPressureBarRetracted;
HMIData.pressureBarService.extendedFeedback := iPressureBarExtended;

autoModeSelected := (_mode = DEVICE_MODES.Auto);
semiAutoModeSelected := (_mode = DEVICE_MODES.SemiAuto);
manualModeSelected := (_mode = DEVICE_MODES.Manual);

timerExtendedDebounce(PT := INT_TO_TIME(extendDelaySP));
timerExtendDwell(PT := INT_TO_TIME(extendDwellSP));
timerRetractedDebounce(PT := INT_TO_TIME(retractDelaySP));
timerRetractDwell(PT := INT_TO_TIME(retractDwellSP));
timerObsSwitchFault(PT := T#100MS);
//Go to idle when enabled
IF enableONS.Q OR resetONS.Q THEN    
    state := PRESSURE_BAR_STATES.Idle;
	_reset := FALSE;
	timerObsSwitchFault.IN := FALSE;
END_IF

IF NOT enable THEN
    state := PRESSURE_BAR_STATES.Idle;
END_IF

_ready := (_mode = DEVICE_MODES.Auto) AND NOT (state = PRESSURE_BAR_STATES.Fault);

faultTimer();

CASE state OF
    
                                    
    PRESSURE_BAR_STATES.Idle :                //Initial state
                                    IF (semiAutoModeSelected AND startCyclePB) OR (autoModeSelected AND _amOpenJaw) OR HMIData.pressureBarService.extendCommand THEN
                                        state := PRESSURE_BAR_STATES.OpenJaw;
                                        _amOpenJaw := FALSE;
										HMIData.pressureBarService.extendCommand := FALSE;
                                    ELSIF (autoModeSelected AND _amCloseJaw) OR HMIData.pressureBarService.retractCommand THEN
                                        state := PRESSURE_BAR_STATES.CloseJaw;
										_amCloseJaw := FALSE;
										HMIData.pressureBarService.retractCommand := FALSE;
                                    ELSIF manualModeSelected THEN
                                        state := PRESSURE_BAR_STATES.Manual;
                                    END_IF
                                    timerObsSwitchFault.IN := FALSE;
    
    PRESSURE_BAR_STATES.OpenJaw :                //Open jaw by extending cylinder
                                    ExtendCylinderHighPressure();
                                    state := PRESSURE_BAR_STATES.OpeningJaw;
    
    PRESSURE_BAR_STATES.OpeningJaw :            //
                                    //This delay is a debounce for the sensors.
                                    faultTimer.PT := T#3S;
									faultTimer.IN := TRUE;
									IF iPressureBarExtended THEN
                                        timerExtendedDebounce.IN := TRUE;
                                        IF timerExtendedDebounce.Q THEN
                                            state := PRESSURE_BAR_STATES.JawOpened;
                                            timerExtendedDebounce.IN := FALSE;
											faultTimer.IN := FALSE;
                                        END_IF
									ELSIF faultTimer.Q THEN
										faultTimer.IN := FALSE;
										faults.failedToOpen.Trigger();
										state := PRESSURE_BAR_STATES.Fault;
                                    END_IF

                                    
                                    
    
    PRESSURE_BAR_STATES.JawOpened :            //Jaw is opened.  If in semi auto mode, go to close jaw after extend dwell. 
                                    IF (semiAutoModeSelected AND startCyclePB) THEN
                                        timerExtendDwell.IN := TRUE;
                                    END_IF
                                    
                                    IF timerExtendDwell.Q OR (autoModeSelected AND _amCloseJaw) OR HMIData.pressureBarService.retractCommand THEN
                                        state := PRESSURE_BAR_STATES.CloseJaw;
                                        _amCloseJaw := FALSE;
										HMIData.pressureBarService.retractCommand := FALSE;
                                        timerExtendDwell.IN := FALSE;
                                    END_IF
    
    PRESSURE_BAR_STATES.CloseJaw :            //Close jaw by retracting cylinder
                                    RetractCylinder();
                                    state := PRESSURE_BAR_STATES.ClosingJaw;
    
    PRESSURE_BAR_STATES.ClosingJaw :            //
                                    //This delay is a debounce after the sensor is seen
                                    faultTimer.PT := T#3S;
									faultTimer.IN := TRUE;
									IF iPressureBarRetracted THEN
                                        timerRetractedDebounce.IN := TRUE;    
                                        IF timerRetractedDebounce.Q THEN
                                            state := PRESSURE_BAR_STATES.JawClosed;
                                            timerRetractedDebounce.IN := FALSE;
											faultTimer.IN := FALSE;
                                        END_IF
									ELSIF faultTimer.Q THEN
										faultTimer.IN := FALSE;
										faults.failedToClose.Trigger();
										ExtendCylinderLowPressure();
										state := PRESSURE_BAR_STATES.Fault;
                                    END_IF
									IF NOT iPressureBarNotObstructed AND NOT iPressureBarRetracted THEN
										faults.obstructionDetected.Trigger();
										ExtendCylinderLowPressure();
										faultTimer.IN := FALSE;
										state := PRESSURE_BAR_STATES.Fault;
									END_IF
                                    
                                    
                                    
    
    PRESSURE_BAR_STATES.JawClosed :            //Go to sealing if seal bar enabled, otherwise if in auto mode go to open jaw after retract dwell. Else go back to idle

                                    
                                    IF (semiAutoModeSelected AND startCyclePB) THEN
                                        timerRetractDwell.IN := TRUE;
                                    END_IF    
									IF iPressureBarNotObstructed THEN
										timerObsSwitchFault.IN := TRUE;
										IF timerObsSwitchFault.Q THEN
											ExtendCylinderLowPressure();
											faults.obstructionFailedToSwitch.Trigger();
											state := PRESSURE_BAR_STATES.Fault;
										END_IF
									ELSE
										timerObsSwitchFault.IN := FALSE;
									END_IF
                                    
                                    IF timerRetractDwell.Q OR (autoModeSelected AND _amOpenJaw) OR HMIData.pressureBarService.extendCommand THEN
                                        state := PRESSURE_BAR_STATES.OpenJaw;
										HMIData.pressureBarService.extendCommand := FALSE;
                                        _amOpenJaw := FALSE;
                                        timerRetractDwell.IN := FALSE;
                                    END_IF

 
    PRESSURE_BAR_STATES.Manual :    IF manualExhaustPB THEN
                                        ExhaustCylinder();
                                        manualExhaustPB := FALSE;
                                    ELSIF manualRetractPB THEN
                                        RetractCylinder();
                                        manualRetractPB := FALSE;
                                    ELSIF manualExtendHighPressurePB THEN
                                        ExtendCylinderHighPressure();
                                        manualExtendHighPressurePB := FALSE;
									ELSIF manualExtendLowPressurePB THEN
                                        ExtendCylinderLowPressure();
                                        manualExtendLowPressurePB := FALSE;
                                    END_IF
                                
    PRESSURE_BAR_STATES.Fault : 
    
END_CASE

IF NOT iPressureBarNotObstructed AND Globals.jawMovingIn THEN
										faults.obstructionDetected.Trigger();
										//ExtendCylinderLowPressure();
										ExhaustCylinder();
										faultTimer.IN := FALSE;
										state := PRESSURE_BAR_STATES.Fault;
END_IF
IF iPressureBarExtended AND iPressureBarRetracted THEN
	faults.sensorFault.Trigger();
END_IF

//Count cycles
incrementCount(CLK :=timerExtendDwell.Q); 
IF incrementCount.Q THEN
    cumulativeHeadCycleCount := cumulativeHeadCycleCount + 1;
END_IF

METHOD AutoSealBag
VAR_INPUT
END_VAR
END_METHOD

METHOD RetractCylinder
VAR_INPUT
END_VAR
oExtendCylinder := FALSE;
oRetractCylinder := TRUE;
END_METHOD

METHOD AutoOpenJaw
VAR_INPUT
END_VAR
_amOpenJaw := TRUE;
END_METHOD

METHOD ExhaustCylinder
VAR_INPUT
END_VAR
oExtendCylinder := FALSE;
oRetractCylinder := FALSE;
END_METHOD

METHOD AutoDoneMovingPassthrough
VAR_INPUT
END_VAR
state := PRESSURE_BAR_STATES.Idle;
END_METHOD

PROPERTY Mode : DEVICE_MODES
SET
_mode := Mode;
END_SET
GET
Mode := _mode;
END_GET
END_PROPERTY

METHOD ExtendCylinderHighPressure
VAR_INPUT
END_VAR
oExtendCylinder := TRUE;
oRetractCylinder := FALSE;
END_METHOD

METHOD AutoCloseJaw
VAR_INPUT
END_VAR
_amCloseJaw := TRUE;
END_METHOD

PROPERTY Ready : BOOL
GET
Ready := _ready;
END_GET
SET
_ready := Ready;
END_SET
END_PROPERTY

METHOD AutoMovingPassthrough
VAR_INPUT
END_VAR
//state := PRESSURE_BAR_STATES.Manual;
state := PRESSURE_BAR_STATES.Idle;
END_METHOD

METHOD ExtendCylinderLowPressure
VAR_INPUT
END_VAR
oExtendCylinder := TRUE;
oRetractCylinder := TRUE;
END_METHOD

END_FUNCTION_BLOCK

// Device/Application/FBs/Temp Sensors/FB_IFMTempSensor
FUNCTION_BLOCK FB_IFMTempSensor EXTENDS FB_TemperatureSensor
VAR_INPUT
	ptrTemperatureBytes : POINTER TO ARRAY[0..1] OF BYTE; 
END_VAR
VAR_OUTPUT
	rtdFailure : FB_Fault(name := 'RTD Failure');
END_VAR
VAR
END_VAR

//	Function Block: FB_IFMTempSensor
//	Description: Implemention of an IFM TP3232 IOLink temperature sensor
//	
//	Created by: Ben Hess
//	Created Date: Tuesday, September 11, 2018

METHOD Execute
VAR_INPUT
END_VAR
_rawTemperatureReading := TO_INT(OSCAT_BASIC.WORD_OF_BYTE(B0 := ptrTemperatureBytes^[1], B1 := ptrTemperatureBytes^[0])); 
_temperatureReadingC := TO_REAL(_rawTemperatureReading / 10.0);
_temperatureReadingF := OSCAT_BASIC.C_TO_F(_temperatureReadingC);

IF _rawTemperatureReading = 0 AND Globals.machinePowerOK THEN 
	rtdFailure.Trigger();
END_IF
END_METHOD

END_FUNCTION_BLOCK

// Device/Application/FBs/Temp Sensors/FB_TemperatureSensor
FUNCTION_BLOCK FB_TemperatureSensor IMPLEMENTS ITempSensor
VAR_INPUT
END_VAR
VAR_OUTPUT
END_VAR
VAR
	_instanceName : STRING;			// Instance Name
	_rawTemperatureReading : INT;   // Raw reading from sensor
	_temperatureReadingC : REAL;	// Scaled temperaure reading in degC
	_temperatureReadingF : REAL;	// Scaled temperaure reading in degF
END_VAR

{attribute 'monitoring' := 'variable'}
PROPERTY TempReadingC : REAL
GET
TempReadingC := _temperatureReadingC;
END_GET
SET
_temperatureReadingC := TempReadingC;
END_SET
END_PROPERTY

{attribute 'monitoring' := 'variable'}
PROPERTY TempReadingF : REAL
GET
TempReadingF := _temperatureReadingF;
END_GET
SET
TempReadingF := _temperatureReadingF;
END_SET
END_PROPERTY

{attribute 'monitoring' := 'variable'}
PROPERTY InstanceName : STRING
GET
InstanceName := _instanceName;
END_GET
END_PROPERTY

END_FUNCTION_BLOCK

// Device/Application/FBs/Temp Sensors/ITempSensor
INTERFACE ITempSensor

PROPERTY TempReadingF : REAL
GET
END_GET
SET
END_SET
END_PROPERTY

PROPERTY TempReadingC : REAL
SET
END_SET
GET
END_GET
END_PROPERTY

END_INTERFACE

// Device/Application/FBs/Temp Sensors/FB_TempController
FUNCTION_BLOCK FB_TempController EXTENDS BaseComponentFB
VAR_INPUT
	temperatureSensor : ITempSensor;
	temperatureSetpoint : REAL;
END_VAR
VAR_OUTPUT
	heaterPulse : BOOL;
	currentTemp : REAL;
	thermalRunawayOvershoot : FB_Fault(name := 'Thermal Runaway - Overshoot');
	thermalRunawayNotHeating : FB_Fault(name := 'Thermal Runaway - Not Heating');
	tempOK : BOOL; // At desired temperature
	cooling : BOOL; // Cooling down to setpoint temp
	heating : BOOL; // Heating up to setpoint temp
END_VAR
VAR
	_manualOutput : REAL;
	_manualMode : BOOL;
	_kp : REAL := 150;
	_ki : REAL := 2;
	_ll : REAL := 0;
	_lh : REAL := 1000;
	_deadBand : REAL := 1;
	_pwmHz : REAL := 1;
	updateTimer : TON := (PT := T#100ms);
	PI : OSCAT_BASIC.CTRL_PI;
	PWM : OSCAT_BASIC.CTRL_PWM;
	tempScaled : DINT;
	diffScaled : DINT;
	diffLast : DINT;
	lastTemp : REAL;
	thermRunawayNHUpdateTimer : Standard.TON := (PT := T#60S);
	thermRunawayNHFaultTimer : Standard.TON := (PT := T#61S);
	thermRunawayOSUpdateTimer : Standard.TON := (PT := T#60S);
	thermRunawayOSFaultTimer : Standard.TON := (PT := T#61S);
END_VAR

SUPER^();
IF enableONS.Q THEN
	lastTemp := currentTemp;
END_IF
updateTimer(IN := NOT updateTimer.Q);
thermRunawayNHUpdateTimer();
thermRunawayNHFaultTimer();
thermRunawayOSUpdateTimer();
thermRunawayOSFaultTimer();

IF updateTimer.Q THEN
	PI(
		ACT:= temperatureSensor.TempReadingF, 
		SET:= temperatureSetpoint, 
		SUP:= _deadBand, 
		OFS:= , 
		M_I:= _manualOutput, 
		MAN:= _manualMode, 
		RST:= , 
		KP:= _kp, 
		KI:= _ki, 
		LL:= _ll, 
		LH:= _lh, 
		Y=> , 
		DIFF=> , 
		LIM=> );

END_IF
cooling := (enable AND temperatureSensor.TempReadingF > temperatureSetpoint) OR NOT enable;
heating := enable AND temperatureSensor.TempReadingF < temperatureSetpoint;
diffScaled := TO_DINT((PI.DIFF * 1000));

diffScaled := TO_DINT((PI.DIFF * 1000));
currentTemp := temperatureSensor.TempReadingF;
tempScaled := TO_DINT((temperatureSensor.TempReadingF * 1000));

PWM(
	CI:= PI.Y / 1000, 
	MAN_IN:= , 
	MANUAL:= , 
	F:= _pwmHz , 
	Q=> heaterPulse);
	
IF NOT enable OR REAL_TO_INT(temperatureSensor.TempReadingC) = 0 THEN
	_manualMode := TRUE;
	_manualOutput := 0.0;
ELSE
	_manualMode := FALSE;
END_IF

// Thermal Runaway - not heating
IF (NOT tempOK AND heating) AND NOT thermalRunawayNotHeating.active THEN
	thermRunawayNHUpdateTimer.IN := TRUE;
	IF thermRunawayNHUpdateTimer.Q THEN
		IF TO_DINT(currentTemp) > TO_DINT(lastTemp) THEN
			thermRunawayNHFaultTimer.IN := FALSE;
		ELSE
			thermRunawayNHFaultTimer.IN := TRUE;
		END_IF
		lastTemp := currentTemp; 
		thermRunawayNHUpdateTimer.IN := FALSE;
	END_IF	
ELSE
	thermRunawayNHUpdateTimer.IN := FALSE;
END_IF

IF thermRunawayNHFaultTimer.Q THEN
	thermalRunawayNotHeating.Trigger();
	thermRunawayNHFaultTimer.IN := FALSE;
END_IF

// Thermal Runaway - overshoot
IF (NOT tempOK AND cooling) AND NOT thermalRunawayOvershoot.active THEN
	thermRunawayOSUpdateTimer.IN := TRUE;
	IF thermRunawayOSUpdateTimer.Q THEN
		IF TO_DINT(currentTemp) < TO_DINT(lastTemp) THEN
			thermRunawayOSFaultTimer.IN := FALSE;
		ELSE
			thermRunawayOSFaultTimer.IN := TRUE;
		END_IF
		lastTemp := currentTemp; 
		thermRunawayOSUpdateTimer.IN := FALSE;
	END_IF	
ELSE
	thermRunawayOSUpdateTimer.IN := FALSE;
END_IF

IF thermRunawayOSFaultTimer.Q THEN
	thermalRunawayOvershoot.Trigger();
	thermRunawayOSFaultTimer.IN := FALSE;
END_IF


IF currentTemp < (temperatureSetpoint - 10) OR currentTemp > (temperatureSetpoint + 10) THEN
	HMIData.sealBarNotAtTemperature.active := TRUE;
	tempOK := FALSE;
ELSE
	HMIData.sealBarNotAtTemperature.active := FALSE;
	tempOK := TRUE;
	lastTemp := currentTemp;
END_IF

IF HMIData.faultActive THEN
	thermRunawayNHUpdateTimer.IN := FALSE;
	thermRunawayNHFaultTimer.IN := FALSE;
	thermRunawayOSUpdateTimer.IN := FALSE;
	thermRunawayOSFaultTimer.IN := FALSE;
END_IF

END_FUNCTION_BLOCK

// Device/Application/FBs/Components/BagDeliveryFB
FUNCTION_BLOCK BagDeliveryFB EXTENDS BaseComponentFB IMPLEMENTS IComponentStatus
VAR_INPUT
    feedBagPB : BOOL;                // Manually Feed bag out
	jogForwardPB : BOOL;
	jogReversePB : BOOL;
    bagsToFeedSetpoint : INT;        // Bags to feed setpoint for testing
    reverseDistanceSetpoint : REAL := -3;  // Distance to reverse
    bagLengthSetpoint : REAL := 23.5;  // Bag length to feed
    accelSetpoint : INT := 600;            // Acceleration Setpoint
    decelSetpoint : INT := 2000;        // Deceleration Setpoint
    reverseVelocitySetpoint : INT := 3;            // Reverse Velocity setoint (IPS)
    feedVelocitySetpoint : INT := 55;            // Bag Feed Velocity setoint (IPS)
    printVelocitySetpoint : UDINT := 6;            // Print speed (IPS)
    sealOffsetSetpoint : REAL := 1.5;            // Seal Offset
    printOffsetSetpoint : REAL := 3;            // Print Offset
    printLengthSetpoint : REAL := 8;                    // Print length
	reverseToPrintHeadSetpoint : REAL := -1.25;
	feedToPhotoeyeSetpoint : REAL := 2.0;
	useLastPrinterDelta : BOOL := TRUE;
	tensionFailONS : FB_ONS;
END_VAR
VAR_OUTPUT
    state : BAG_DELIVERY_STATES;    // Current state of bag delivery component
	reverseFault : FB_Fault(name := 'Reverse Fault');
	noBagOverEye : FB_Fault(name := 'No bag over Photoeye');
	bagTensionFault : FB_Fault(name := 'Bag Tension Fault');
END_VAR
VAR
    delay : TON := (PT := T#100MS);    // Delay for testing
	jogForwardONS: FB_ONS;
	jogReverseONS: FB_ONS;
	delayForReverseFault : Standard.TON;
	autoFeedDelay : TON := (PT := T#200MS);
	sealBarToPrintHeadLength : REAL;
    bagsCurrentlyFed  :INT;            // Bags currently fed for testing
    remainingLength : REAL;            // Remaining bag length after print
	delayForPrintFeed : TIME := T#20MS;
	printerExtraFeedLength : REAL := 0.25;
    //bagFeedMasterMotor : FB_AppliedMotionStepServoTCP();
    //bagFeedMasterMotor : FB_AppliedMotionBagDeliveryMotor();
	bagFeedMasterMotor : FB_AppliedMotionBagDeliveryMotor_1();
	bagFeedRearMotor : FB_AppliedMotionBagDeliveryMotor_1();
	accelPercent : REAL := 0.1;
	decelPercent : REAL := 0.05;
    _amReverseBag : BOOL;            // Auto Mode - Reverse bag
    _amFeedBagOut : BOOL;            // Auto Mode - Feed new bag out
    _amWaitForPrinter : BOOL;        // Auto Mode - wait for printer
    _amPrinterReady : BOOL;            // Auto Mode - Printer is ready
    _amStartPrint : BOOL;            // Auto Mode - Start Printing
    _amPrinterDone : BOOL;             // Auto Mode - Printer is Done
	_amFeedToEye : BOOL;			  // Auto Mode - Feed Bag to Eye
	testTorque : BOOL;
	testTorqueValue : DINT := 60;
	reverseSpeedDistanceOffset : REAL;
END_VAR

//    Function Block: BagDeliveryFB
//    Description: This is the state machine for the bag delivery test rig
//    
//    Created by: Ben Hess
//    Created Date: Thursday, April 19, 2018

SUPER^();
tensionFailONS(CLK := iBagTensionFault);
reverseSpeedDistanceOffset := OSCAT_BASIC.SCALE_R(HMIData.bagReverseSpeed,3,10,0,0.5);
reverseToPrintHeadSetpoint := -1.75 + reverseSpeedDistanceOffset;
delay();
delayForReverseFault();
autoFeedDelay(IN := _amFeedBagOut);

bagLengthSetpoint := HMIData.bagLength;
printVelocitySetpoint := HMIData.printSpeed;
sealOffsetSetpoint := HMIData.bagSkirtLength;
printOffsetSetpoint := HMIData.printOffset;
sealBarToPrintHeadLength := ABS(reverseToPrintHeadSetpoint) + 2.25;
printLengthSetpoint := HMIData.printLength;
reverseVelocitySetpoint := TO_INT(HMIData.bagReverseSpeed);
feedVelocitySetpoint := TO_INT(HMIData.bagForwardSpeed);
IF HMIData.baggerModelSelection = ModelSelection.Pro18 THEN
	reverseToPrintHeadSetpoint := -1.25;
ELSE
	reverseToPrintHeadSetpoint := -1.0;
END_IF


(*bagFeedMasterMotor(modbusInputParameters := BagDeliverMasterMotorModbusInputs, 
                    stepsPerInchSetpoint := Globals.STEPS_PER_INCH_20_DEGREE_BAG_DELIVERY, 
                    reversePolarity := FALSE, 
                    slave := Bag_Delivery_Master_Motor);*)
bagFeedMasterMotor(ptrEIPInputs := ADR(bagDeliveryMotorInputs),
                ptrEIPOutputs := ADR(bagDeliveryMotorOutputs),
                stepsPerInchSetpoint := Globals.STEPS_PER_INCH_PRO24_BAG_DELIVERY,
                //faultHandler := PRG_Bagger.faultHandler,
				reversePolarity := FALSE, 
				defaultCurrentSetpoint := 1150, 
				commFail := Bag_Delivery_EIP_Motor.udiState <> 4);
bagFeedMasterMotor.Execute();

bagFeedRearMotor(ptrEIPInputs := ADR(bagRearMotorInputs),
                ptrEIPOutputs := ADR(bagRearMotorOutputs),
                stepsPerInchSetpoint := Globals.STEPS_PER_INCH_PRO24_BAG_DELIVERY,
                //faultHandler := PRG_Bagger.faultHandler,
				reversePolarity := FALSE, 
				defaultCurrentSetpoint := 1150, 
				commFail := Bag_Delivery_Rear_Motor.udiState <> 4);
bagFeedRearMotor.Execute();

IF testTorque THEN
	//bagFeedRearMotor.SetRearMotorTorqueValue(testTorqueValue);
	testTorque := FALSE;
END_IF

IF enableONS.Q OR resetONS.Q THEN
    IF _mode = DEVICE_MODES.Manual THEN 
        state := BAG_DELIVERY_STATES.Manual;
    ELSE
        state := BAG_DELIVERY_STATES.Idle;
    END_IF
	_reset := FALSE;
	ClearCommands();
END_IF
jogForwardONS(CLK := jogForwardPB);
jogReverseONS(CLK := jogReversePB);
IF NOT enable THEN
    state := BAG_DELIVERY_STATES.Idle;
END_IF
delay();
_ready := (_mode = DEVICE_MODES.Auto) AND (NOT (state = BAG_DELIVERY_STATES.Fault) OR NOT (state = BAG_DELIVERY_STATES.Idle));

IF tensionFailONS.OSR AND NOT Globals.enableDryCycle THEN
	bagTensionFault.Trigger();
END_IF

CASE state OF
    BAG_DELIVERY_STATES.Idle :                     
													IF _mode = DEVICE_MODES.Manual THEN 
														state := BAG_DELIVERY_STATES.Manual;
													ELSIF NOT iBagNotPresent OR Globals.enableDryCycle THEN
														state := BAG_DELIVERY_STATES.Ready;
													//ELSIF iBagNotPresent AND (_amFeedToEye OR _amReverseBag) THEN
													ELSIF (_amFeedToEye OR _amReverseBag) THEN
														state := BAG_DELIVERY_STATES.FeedToEye;
														_amFeedToEye := FALSE;
													END_IF
													IF jogForwardONS.OSR THEN
														bagFeedMasterMotor.MoveDistance(distance := 30, 
                                                                                    acceleration := accelSetpoint, 
                                                                                    deceleration := decelSetpoint, 
                                                                                    velocity := REAL_TO_INT((1 * Globals.VELOCITY_IPS_MULTIPLIER_20_DEGREE_BAG_DELIVERY)));
													ELSIF jogReverseONS.OSR THEN
														bagFeedMasterMotor.MoveDistance(distance := -30, 
                                                                                    acceleration := accelSetpoint, 
                                                                                    deceleration := decelSetpoint, 
                                                                                    velocity := REAL_TO_INT((1 * Globals.VELOCITY_IPS_MULTIPLIER_20_DEGREE_BAG_DELIVERY)));
													ELSIF jogForwardONS.OSF OR jogReverseONS.OSF THEN
														bagFeedMasterMotor.Stop();
													END_IF
    
	BAG_DELIVERY_STATES.FeedToEye :					//Feed to photoeye if not present
													IF iBagNotPresent THEN
														bagFeedMasterMotor.MoveDistance(distance := feedToPhotoeyeSetpoint, 
                                                                                    acceleration := accelSetpoint, 
                                                                                    deceleration := decelSetpoint, 
                                                                                    velocity := REAL_TO_INT((feedToPhotoeyeSetpoint * Globals.VELOCITY_IPS_MULTIPLIER_20_DEGREE_BAG_DELIVERY)));
														state := BAG_DELIVERY_STATES.FeedingToEye;
													ELSE
														state := BAG_DELIVERY_STATES.SetTorqueMode;
													END_IF
													
													
	BAG_DELIVERY_STATES.FeedingToEye :				// Stop once photoeye seen
													delay.PT := T#3S;
													delay.IN := TRUE;
													IF NOT iBagNotPresent THEN
														bagFeedMasterMotor.Stop();
														state := BAG_DELIVERY_STATES.SetTorqueMode;
														delay.IN := FALSE;
													END_IF
													IF delay.Q THEN
														state := BAG_DELIVERY_STATES.Fault;
														noBagOverEye.Trigger();
														delay.IN := FALSE;
													END_IF
	
	BAG_DELIVERY_STATES.SetTorqueMode :				// Set torque following mode
													delay.PT := T#50MS;
													delay.IN := TRUE;
													IF delay.Q THEN
														bagFeedMasterMotor.SetRearMotorToTorqueMode();
														state := BAG_DELIVERY_STATES.Idle;	
														delay.IN := FALSE;
													END_IF
													
	
    BAG_DELIVERY_STATES.Reverse :                    // Reverse to break perf
                                                    bagFeedMasterMotor.MoveDistance(distance := reverseDistanceSetpoint, 
                                                                                    acceleration := TO_INT((ABS(reverseDistanceSetpoint) * Globals.STEPS_PER_INCH_20_DEGREE_BAG_DELIVERY) *  accelPercent),
                                                                                    deceleration := TO_INT((ABS(reverseDistanceSetpoint) * Globals.STEPS_PER_INCH_20_DEGREE_BAG_DELIVERY) *  decelPercent), 
                                                                                    velocity := REAL_TO_INT((reverseVelocitySetpoint * Globals.VELOCITY_IPS_MULTIPLIER_20_DEGREE_BAG_DELIVERY)));    
                                                        state := BAG_DELIVERY_STATES.Reversing;
                                                    
                                                    
    BAG_DELIVERY_STATES.Reversing :                    // Back up until we see the trailing edge of the bag
														 IF iBagNotPresent OR Globals.enableDryCycle THEN
															delay.PT := T#10MS;
															delay.IN := TRUE;
															IF delay.Q THEN
																bagFeedMasterMotor.Stop();
																delay.IN := FALSE;
																delayForReverseFault.IN := FALSE;
																state := BAG_DELIVERY_STATES.ReverseToPrinthead;
															END_IF
														ELSIF bagFeedMasterMotor.CommandAcknowledged AND NOT iBagNotPresent THEN
															delayForReverseFault.PT := T#3000MS;
															delayForReverseFault.IN := TRUE;
															IF delayForReverseFault.Q THEN
																reverseFault.Trigger();
																bagFeedMasterMotor.Stop();
															delayForReverseFault.IN := FALSE;
															state := BAG_DELIVERY_STATES.Fault; 
															END_IF
															
														END_IF
											
                                                  
													
	BAG_DELIVERY_STATES.ReverseToPrinthead :                    // Reverse to print head
                                                    delay.PT := T#50MS;
													delay.IN := TRUE;
													IF delay.Q THEN
														bagFeedMasterMotor.MoveDistanceFinal(distance := reverseToPrintHeadSetpoint, 
                                                                                    acceleration := TO_INT((ABS(reverseToPrintHeadSetpoint) * Globals.STEPS_PER_INCH_20_DEGREE_BAG_DELIVERY) *  accelPercent),
                                                                                    deceleration := TO_INT((ABS(reverseToPrintHeadSetpoint) * Globals.STEPS_PER_INCH_20_DEGREE_BAG_DELIVERY) *  decelPercent), 
                                                                                    velocity := REAL_TO_INT((reverseVelocitySetpoint * Globals.VELOCITY_IPS_MULTIPLIER_20_DEGREE_BAG_DELIVERY)));    
                                                    	state := BAG_DELIVERY_STATES.ReversingToPrintHead;
														delay.IN := FALSE;
													END_IF
													
													
	BAG_DELIVERY_STATES.ReversingToPrintHead :                    // Reverse to break perf
                                                   	delay.PT := T#50MS;
													delay.IN := TRUE;
													
													IF delay.Q THEN
														IF bagFeedMasterMotor.CommandAcknowledged AND bagFeedMasterMotor.InPosition THEN
                                                        	state := BAG_DELIVERY_STATES.ReverseDone;
                                                    	END_IF
														delay.IN := FALSE;
													END_IF
                                                    
    BAG_DELIVERY_STATES.ReverseDone :                // We don't print in semi auto or manual mode.  In auto mode if the printer is selected then we move to those states
                                                    IF _mode = DEVICE_MODES.SemiAuto OR _mode = DEVICE_MODES.Manual OR (_mode  = DEVICE_MODES.Auto AND autoFeedDelay.Q) THEN
                                                        IF bagFeedMasterMotor.CommandAcknowledged THEN
															state := BAG_DELIVERY_STATES.FeedBagOut;
                                                        	remainingLength := bagLengthSetpoint;
                                                        	_amFeedBagOut := FALSE;
														END_IF
														
                                                    ELSIF (_mode  = DEVICE_MODES.Auto AND _amWaitForPrinter) THEN
                                                        IF bagFeedMasterMotor.CommandAcknowledged THEN
															state := BAG_DELIVERY_STATES.WaitingForPrinter;
															remainingLength := bagLengthSetpoint - (printLengthSetpoint + printOffsetSetpoint + printerExtraFeedLength);
															_amWaitForPrinter := FALSE;  
														END_IF  
                                                    END_IF
                                                        
                                                    
    BAG_DELIVERY_STATES.WaitingForPrinter :            // 
                                                    IF (_mode  = DEVICE_MODES.Auto AND _amPrinterReady) THEN
														IF printOffsetSetpoint <> 0 THEN
															state := BAG_DELIVERY_STATES.FeedToPrintOffset;
														ELSE
															state := BAG_DELIVERY_STATES.FedToPrintOffset;
														END_IF
                                                        
                                                        _amPrinterReady := FALSE;
                                                    END_IF
                                                        
    BAG_DELIVERY_STATES.FeedToPrintOffset :            // 
                                                    bagFeedMasterMotor.MoveDistance(distance := printOffsetSetpoint, 
                                                                                    acceleration := accelSetpoint, 
                                                                                    deceleration := decelSetpoint, 
                                                                                    velocity := REAL_TO_INT((feedVelocitySetpoint * Globals.VELOCITY_IPS_MULTIPLIER_20_DEGREE_BAG_DELIVERY)));    
                                                        state := BAG_DELIVERY_STATES.FeedingToPrintOffset;
                                                    
    BAG_DELIVERY_STATES.FeedingToPrintOffset :        // 
													delay.PT := T#50MS;
													delay.IN := TRUE;
													
													IF delay.Q THEN
														IF bagFeedMasterMotor.CommandAcknowledged AND bagFeedMasterMotor.InPosition THEN
                                                        	state := BAG_DELIVERY_STATES.FedToPrintOffset;
                                                    	END_IF
														delay.IN := FALSE;
													END_IF
                                                    
                                                    
    BAG_DELIVERY_STATES.FedToPrintOffset :            // 
                                                    IF (_mode  = DEVICE_MODES.Auto AND _amStartPrint) THEN
                                                        state := BAG_DELIVERY_STATES.FeedAtPrintSpeed;
                                                        _amStartPrint := FALSE;
                                                    END_IF
                                                    
    BAG_DELIVERY_STATES.FeedAtPrintSpeed :            // 
													delay.PT := delayForPrintFeed;
                                                    delay.IN := TRUE;
													
													IF delay.Q THEN
														bagFeedMasterMotor.MoveDistance(distance := printLengthSetpoint + printerExtraFeedLength, 
                                                                                    acceleration := accelSetpoint, 
                                                                                    deceleration := decelSetpoint, 
                                                                                    velocity := REAL_TO_INT((printVelocitySetpoint * Globals.VELOCITY_IPS_MULTIPLIER_20_DEGREE_BAG_DELIVERY)));    
                                                        state := BAG_DELIVERY_STATES.FeedingAtPrintSpeed;
														delay.IN := FALSE;
													END_IF
                                                    
    BAG_DELIVERY_STATES.FeedingAtPrintSpeed :        // 
													delay.PT := T#50MS;
													delay.IN := TRUE;
													IF delay.Q THEN
														IF bagFeedMasterMotor.CommandAcknowledged AND bagFeedMasterMotor.InPosition THEN
                                                        	state := BAG_DELIVERY_STATES.FedAtPrintSpeed;
                                                    	END_IF
														delay.IN := FALSE;
													END_IF
                                                   
                                                    
    BAG_DELIVERY_STATES.FedAtPrintSpeed :            // 
                                                    IF (_mode  = DEVICE_MODES.Auto AND _amPrinterDone) THEN
                                                        state := BAG_DELIVERY_STATES.FeedBagOut;
                                                        _amPrinterDone := FALSE;
                                                    END_IF
                                                    
    BAG_DELIVERY_STATES.FeedBagOut :                // Feed bag length out
                                                    //bagFeedMasterMotor.MoveDistanceFinal(distance := (remainingLength + sealOffsetSetpoint + (reverseToPrintHeadSetpoint*-1)), 
													bagFeedMasterMotor.MoveDistanceFinal(distance := (remainingLength + sealBarToPrintHeadLength) - sealOffsetSetpoint, 
                                                                                        acceleration := accelSetpoint, 
                                                                                        deceleration := decelSetpoint, 
                                                                                        velocity := REAL_TO_INT((feedVelocitySetpoint * Globals.VELOCITY_IPS_MULTIPLIER_20_DEGREE_BAG_DELIVERY)));
                                                    state := BAG_DELIVERY_STATES.FeedingBagOut;    
    
    BAG_DELIVERY_STATES.FeedingBagOut :                // Wait until move is done
													delay.PT := T#50MS;
													delay.IN := TRUE;
													IF delay.Q THEN
														IF bagFeedMasterMotor.CommandAcknowledged AND bagFeedMasterMotor.InPosition THEN
                                                        state := BAG_DELIVERY_STATES.FedBagOut;
														
                                                    	END_IF
														delay.IN := FALSE;
													END_IF
                                                    
    
    BAG_DELIVERY_STATES.FedBagOut :                    // Go to the next ready state
                                                    IF _mode = DEVICE_MODES.Manual THEN 
                                                        state := BAG_DELIVERY_STATES.Manual;
                                                    ELSE
                                                        state := BAG_DELIVERY_STATES.Ready;
                                                    END_IF
													HMIData.driveRollerClean.SetCount(HMIData.driveRollerClean.count + TO_INT(bagLengthSetpoint));
                                                    Globals.bagDeliveryCycleCount := Globals.bagDeliveryCycleCount + 1;
    
    BAG_DELIVERY_STATES.Ready :                        IF (_mode = DEVICE_MODES.Auto AND _amReverseBag) OR _mode = DEVICE_MODES.SemiAuto THEN 
                                                        state := BAG_DELIVERY_STATES.Reverse;
                                                        ClearCommands();
                                                    END_IF 
													IF _amFeedToEye THEN
														state := BAG_DELIVERY_STATES.SetTorqueMode;
													END_IF
													_amFeedToEye := FALSE;
													IF iBagNotPresent AND NOT Globals.enableDryCycle THEN 
														state := BAG_DELIVERY_STATES.Idle;
													END_IF
													IF jogForwardONS.OSR THEN
														bagFeedMasterMotor.MoveDistance(distance := 30, 
                                                                                    acceleration := accelSetpoint, 
                                                                                    deceleration := decelSetpoint, 
                                                                                    velocity := REAL_TO_INT((1 * Globals.VELOCITY_IPS_MULTIPLIER_20_DEGREE_BAG_DELIVERY)));
													ELSIF jogReverseONS.OSR THEN
														bagFeedMasterMotor.MoveDistance(distance := -30, 
                                                                                    acceleration := accelSetpoint, 
                                                                                    deceleration := decelSetpoint, 
                                                                                    velocity := REAL_TO_INT((1 * Globals.VELOCITY_IPS_MULTIPLIER_20_DEGREE_BAG_DELIVERY)));
													ELSIF jogForwardONS.OSF OR jogReverseONS.OSF THEN
														bagFeedMasterMotor.Stop();
													END_IF
    
    BAG_DELIVERY_STATES.Fault :                        ClearCommands();
													IF jogForwardONS.OSR THEN
														bagFeedMasterMotor.MoveDistance(distance := 30, 
                                                                                    acceleration := accelSetpoint, 
                                                                                    deceleration := decelSetpoint, 
                                                                                    velocity := REAL_TO_INT((1 * Globals.VELOCITY_IPS_MULTIPLIER_20_DEGREE_BAG_DELIVERY)));
													ELSIF jogReverseONS.OSR THEN
														bagFeedMasterMotor.MoveDistance(distance := -30, 
                                                                                    acceleration := accelSetpoint, 
                                                                                    deceleration := decelSetpoint, 
                                                                                    velocity := REAL_TO_INT((1 * Globals.VELOCITY_IPS_MULTIPLIER_20_DEGREE_BAG_DELIVERY)));
													ELSIF jogForwardONS.OSF OR jogReverseONS.OSF THEN
														bagFeedMasterMotor.Stop();
													END_IF
    
    BAG_DELIVERY_STATES.Manual :                    IF _mode = DEVICE_MODES.Auto THEN
														state := BAG_DELIVERY_STATES.Ready;	
													END_IF
													// Manually feed bags out
                                                    IF feedBagPB THEN
                                                        state := BAG_DELIVERY_STATES.Reverse;
                                                        feedBagPB := FALSE;
                                                    END_IF
                                                        
END_CASE

METHOD AutoPrinterDone
VAR_INPUT
END_VAR
_amPrinterDone := TRUE;
END_METHOD

METHOD AutoFeedToEye
VAR_INPUT
END_VAR
_amFeedToEye := TRUE;
END_METHOD

METHOD AutoWaitForPrinter
VAR_INPUT
END_VAR
_amWaitForPrinter := TRUE;
END_METHOD

METHOD AutoReverseBag
VAR_INPUT
END_VAR
_amReverseBag := TRUE;
END_METHOD

METHOD PRIVATE ClearCommands
VAR_INPUT
END_VAR
_amFeedBagOut := FALSE;
_amReverseBag := FALSE;
_amPrinterDone := FALSE;
_amPrinterReady := FALSE;
_amWaitForPrinter := FALSE;
_amStartPrint := FALSE;
//_amFeedToEye := FALSE;
END_METHOD

METHOD AutoPrinterReady
VAR_INPUT
END_VAR
_amPrinterReady := TRUE;
END_METHOD

PROPERTY Mode : DEVICE_MODES
GET
Mode := _mode;
END_GET
SET
_mode := Mode;
END_SET
END_PROPERTY

PROPERTY Ready : BOOL
SET
_ready := Ready;
END_SET
GET
Ready := _ready;
END_GET
END_PROPERTY

METHOD AutoFeedBagOut
VAR_INPUT
END_VAR
_amFeedBagOut := TRUE;
END_METHOD

METHOD AutoStartPrintFeed
VAR_INPUT
END_VAR
_amStartPrint := TRUE;
END_METHOD

END_FUNCTION_BLOCK

// Device/Application/FBs/Motors/Applied Motion/FB_AppliedMotionStepServoTCP
FUNCTION_BLOCK FB_AppliedMotionStepServoTCP EXTENDS FB_AppliedMotionStepServoMBBase IMPLEMENTS IPositionableMotor
VAR_INPUT
END_VAR
VAR_IN_OUT
    slave : IoDrvModbusTCP.ModbusTCPSlave;                    //Slave ModbusTCP Object
END_VAR
VAR_OUTPUT
END_VAR
VAR
    sendMoveCommand : FB_SendMoveCommandAppliedMotionTCP();
    sendOpcodeCommand :  FB_SendOpcodeCommandAppliedMotionTCP();
END_VAR

sendMoveCommand(Slave := slave);
sendOpcodeCommand(Slave := slave);

commandSuccessful S= (sendMoveCommand.xDone OR sendOpcodeCommand.xDone) AND NOT status.inPosition;

METHOD Stop
commandSuccessful := FALSE;
SendOpcodeCommand.opcode := STEP_SERVO_OPCODES.STOP_MOVE_KILL_BUFFER;
SendOpcodeCommand.Execute();
END_METHOD

METHOD MoveToPosition
VAR_INPUT
    (*Position to move to in inches*)
    position    : REAL;
    (*Acceleration in RPM/sec*)
    acceleration    : INT;
    (*Deceleration in RPM/sec*)
    deceleration    : INT;
    (*Velocity in .25RPM*)
    velocity    : INT;
END_VAR
//This method preps the data to send to the drive and triggers the send.
//Set distance and unpack to prep data to send to motor
distanceToMoveInSteps.rawValue := REAL_TO_DINT((position) * stepsPerInchSetpoint);
IF reversePolarity THEN
    distanceToMoveInSteps.rawValue := distanceToMoveInSteps.rawValue * -1;    
END_IF
commandSuccessful := FALSE;
ModbusLongHandler.Unpack(distanceToMoveInSteps);
sendMoveCommand.acceleration := acceleration;
sendMoveCommand.deceleration := deceleration;
sendMoveCommand.velocity := velocity;
sendMoveCommand.distanceHighWord := distanceToMoveInSteps.highWord;
sendMoveCommand.distanceLowWord := distanceToMoveInSteps.lowWord;
sendMoveCommand.opcode := STEP_SERVO_OPCODES.FEED_TO_POSITION;
sendMoveCommand.Execute();
END_METHOD

METHOD ExecuteStoredProgram
VAR_INPUT
    (*Program number to execute*)
    programNumber    : INT;
END_VAR
//Load program into queue by setting it as parameter 1 and send it and the execute queue opcode
commandSuccessful := FALSE;
SendOpcodeCommand.opcode := STEP_SERVO_OPCODES.QUEUE_LOAD_AND_EXECUTE;
SendOpcodeCommand.Parameter1 := INT_TO_WORD(programNumber);
SendOpcodeCommand.Execute();
END_METHOD

METHOD MoveDistance
VAR_INPUT
    distance : REAL;        //Distance to move in inches
    acceleration : INT;        //Acceleration in RPM/sec
    deceleration : INT;        //Deceleration in RPM/sec
    velocity : INT;            //Velocity in .25RPM
END_VAR
//This method preps the data to send to the drive and triggers the send.
//Set distance and unpack to prep data to send to motor
distanceToMoveInSteps.rawValue := REAL_TO_DINT((distance) * stepsPerInchSetpoint);
IF reversePolarity THEN
    distanceToMoveInSteps.rawValue := distanceToMoveInSteps.rawValue * -1;    
END_IF
commandSuccessful := FALSE;
ModbusLongHandler.Unpack(distanceToMoveInSteps);
sendMoveCommand.acceleration := acceleration;
sendMoveCommand.deceleration := deceleration;
sendMoveCommand.velocity := velocity;
sendMoveCommand.distanceHighWord := distanceToMoveInSteps.highWord;
sendMoveCommand.distanceLowWord := distanceToMoveInSteps.lowWord;
sendMoveCommand.opcode := STEP_SERVO_OPCODES.FEED_TO_LENGTH;
sendMoveCommand.Execute();
END_METHOD

METHOD HomeNow
//Load program 1 into queue by setting it as parameter 1 and send it and the execute queue opcode
ExecuteStoredProgram(QX_PROGRAMS.HOME_HARD_STOP);
HomeRequired := FALSE;
END_METHOD

END_FUNCTION_BLOCK

// Device/Application/FBs/Motors/Applied Motion/FB_AppliedMotionStepServoMBBase
FUNCTION_BLOCK FB_AppliedMotionStepServoMBBase IMPLEMENTS IPositionableMotor, IStoredProgramMotor
VAR_INPUT
    modbusInputParameters : ARRAY[0 .. 124] OF WORD;        //This is the input array of words of raw Modbus registers
    stepsPerInchSetpoint : INT;                                        //Steps per inch setpoint
    reversePolarity : BOOL;                                    //0 = Normal, 1 = reversed polarity for display
    pointToPointAccelSetpoint : INT;        //Point-to-Point Acceleration (AC) Setpoint
    pointToPointDecelSetpoint : INT;        //Point-to-Point Deceleration (DE) Setpoint
    velocitySetpoint : INT;                //Velocity (VE) Setpoint
    distanceSetpointInches : REAL;        //Distance setpoint in inches Setpoint
    moveDistanceManualPB : BOOL;            //Move distance pushbutton
    movePositionManualPB : BOOL;            //Move position pushbutton
END_VAR
VAR_IN_OUT
    //slave : IoDrvModbusTCP.ModbusTCPSlave;                    //Slave ModbusTCP Object
END_VAR
VAR
    ModbusLongHandler : ModbusLongHandlerFB();
    absolutePositionSteps : ModbusLongType; //Immediate Absolute Position in steps
    distanceSteps : ModbusLongType;    //Point-to-Point Distance (DI) Input from Drive Combined
    distanceToMoveInSteps : ModbusLongType;        //Distance Setpoint to Drive
    stepServoStatusRaw : INT; //Raw step servo status over modbus
    commandSuccessful : BOOL;    //Modbus Command was successful
    homeRequiredIndication : BOOL; //Home required indication.
    //commandAcked : BOOL;        //Command acked from "send" function blocks
    interfaceToPass : IFault;
    faultListRegisterSuccess : BOOL;        // Registering in fault list successful
    _faulted : BOOL;                    // Motor Faulted
END_VAR
VAR_OUTPUT
    absolutePositonInches : REAL; //Immediate Absolute Positon in inches
    distanceInches : REAL;            //Distance from Drive converted to inches
    homeAccel : INT;    //Home Acceleration (HA) Input from Drive
    homeCurrentLimit : INT;    //Home Hard Stop current limit (HC) Input from Drive
    homeDecel : INT;    //Home Deceleration (HL) Input from Drive
    homeVelocity : INT;    //Home Speed (HV) from Drive
    jogAccel : INT;    //Jog Acceleration (AC) Input from Drive
    jogDecel : INT;    //Jog Deceleration (DE) Input from Drive
    jogVelocity : INT;    //Jog Speed from Drive
    pointToPointAccel : INT;    //Point-to-Point Acceleration (AC) Input from Drive
    pointToPointDecel : INT;    //Point-to-Point Deceleration (DE) Input from Drive
    velocity : INT;    //Velocity (VE) Input from Drive
    status : StepServoStatusFB; //Status of servo
    QSegmentRunning : INT; //Current Q program running from Drive
END_VAR

METHOD Execute
VAR_INPUT
END_VAR
//    Function Block: AppliedMotionStepServo
//    Description: This block provides an abstraction for a Applied Motion Step Servo
//    Created by: Ben Hess
//    Created Date: April 2nd, 2018

//Map raw Modbus Registers to parameters
absolutePositionSteps.highWord := modbusInputParameters[6];
absolutePositionSteps.lowWord := modbusInputParameters[7];
distanceSteps.highWord := modbusInputParameters[30];
distanceSteps.lowWord := modbusInputParameters[31];
jogAccel := WORD_TO_INT(modbusInputParameters[46]);
jogDecel := WORD_TO_INT(modbusInputParameters[47]);
jogVelocity := WORD_TO_INT(modbusInputParameters[48]);
pointToPointAccel := WORD_TO_INT(modbusInputParameters[27]);
pointToPointDecel := WORD_TO_INT(modbusInputParameters[28]);
velocity := WORD_TO_INT(modbusInputParameters[29]);
stepServoStatusRaw := WORD_TO_INT(modbusInputParameters[1]);
QSegmentRunning := WORD_TO_INT(modbusInputParameters[17]);

//Convert Distance setpoint to steps.  Reverse polarity for display purposes if needed. 
//oDistanceSteps.displayValue := REAL_TO_DINT((oDistanceInches) * stepsPerInch);
//oDistanceSteps.rawValue := REAL_TO_DINT((oDistanceInches ) * stepsPerInch);
//DistanceSteps.displayValue := DistanceSteps.rawValue;
distanceInches := (DINT_TO_REAL(distanceSteps.displayValue) / INT_TO_REAL(stepsPerInchSetpoint));    
absolutePositionSteps.displayValue := absolutePositionSteps.rawValue;
absolutePositonInches := (DINT_TO_REAL(absolutePositionSteps.displayValue) / INT_TO_REAL(stepsPerInchSetpoint));

//Homing required from motor - for now just if there was an initialization seen.
homeRequiredIndication S= status.initializing OR Globals.firstScan;

IF reversePolarity THEN
    //oDistanceSteps.rawValue := oDistanceSteps.rawValue * -1; 
    distanceInches := distanceInches * -1;
    absolutePositonInches := absolutePositonInches * -1; 
END_IF

//Get Servo Status and unpack
status(statusCode := StepServoStatusRaw);

//Bit-packing for LONG types over Modbus
ModbusLongHandler.Pack(distanceSteps);
ModbusLongHandler.Pack(absolutePositionSteps);


//Manual moves for motor
IF moveDistanceManualPB THEN
    MoveDistance(distance := distanceSetpointInches, acceleration := pointToPointAccelSetpoint, deceleration := pointToPointDecelSetpoint, velocity := velocitySetpoint);
    moveDistanceManualPB := FALSE;
END_IF

IF movePositionManualPB THEN
    MoveToPosition(position := distanceSetpointInches, acceleration := pointToPointAccelSetpoint, deceleration := pointToPointDecelSetpoint, velocity := velocitySetpoint);
    movePositionManualPB := FALSE;
END_IF
END_METHOD

{attribute 'monitoring' := 'variable'}
PROPERTY HomeRequired : BOOL
SET
homeRequiredIndication := HomeRequired;
END_SET
GET
HomeRequired := homeRequiredIndication;
END_GET
END_PROPERTY

{attribute 'monitoring' := 'variable'}
PROPERTY CommandAcknowledged : BOOL
GET
CommandAcknowledged := commandSuccessful;
END_GET
END_PROPERTY

METHOD ExecuteStoredProgram
VAR_INPUT
    (*Program number to execute*)
    programNumber    : INT;
END_VAR
END_METHOD

{attribute 'monitoring' := 'variable'}
PROPERTY ActiveStoredProgramNumber : INT
GET
ActiveStoredProgramNumber := QSegmentRunning;
END_GET
END_PROPERTY

//{warning 'add method implementation '}
METHOD MoveDistance
VAR_INPUT
    (*Distance to move in inches*)
    distance    : REAL;
    (*Acceleration in RPM/sec*)
    acceleration    : INT;
    (*Deceleration in RPM/sec*)
    deceleration    : INT;
    (*Velocity in .25RPM*)
    velocity    : INT;
END_VAR
END_METHOD

{attribute 'monitoring' := 'variable'}
PROPERTY InPosition : BOOL
GET
InPosition := status.inPosition;
END_GET
END_PROPERTY

METHOD HomeNow
END_METHOD

//{warning 'add method implementation '}
METHOD Stop
END_METHOD

{attribute 'monitoring' := 'variable'}
PROPERTY Homing : BOOL
GET
Homing := status.homing;
END_GET
END_PROPERTY

{attribute 'monitoring' := 'variable'}
PROPERTY CurrentPosition : REAL  //Current motor position in Inches
GET
CurrentPosition := absolutePositonInches;
END_GET
END_PROPERTY

{attribute 'monitoring' := 'variable'}
PROPERTY Moving : BOOL
GET
Moving := status.moving;
END_GET
END_PROPERTY

//{warning 'add method implementation '}
METHOD MoveToPosition
VAR_INPUT
    (*Position to move to in inches*)
    position    : REAL;
    (*Acceleration in RPM/sec*)
    acceleration    : INT;
    (*Deceleration in RPM/sec*)
    deceleration    : INT;
    (*Velocity in .25RPM*)
    velocity    : INT;
END_VAR
END_METHOD

END_FUNCTION_BLOCK

// Device/Application/FBs/DataHandlers/ModbusLongHandlerFB
FUNCTION_BLOCK ModbusLongHandlerFB
VAR_INPUT
    modbusLong : ModbusLongType;
END_VAR
VAR_OUTPUT
END_VAR
VAR
END_VAR

METHOD PackDirect : ModbusLongType
VAR_INPUT
    highWord : WORD;
    lowWord : WORD
;END_VAR
PackDirect.rawValue :=  DWORD_TO_DINT(OSCAT_BASIC.DWORD_OF_WORD(highWord,lowWord));
END_METHOD

METHOD Pack
VAR_IN_OUT
    modbusLong : ModbusLongType;
END_VAR
modbusLong.rawValue := DWORD_TO_DINT(OSCAT_BASIC.DWORD_OF_WORD(modbusLong.highWord,modbusLong.lowWord));
END_METHOD

METHOD Unpack
VAR_IN_OUT
    modbusLong : ModbusLongType;
END_VAR
modbusLong.highWord := OSCAT_BASIC.WORD_OF_DWORD(in := DINT_TO_DWORD(modbusLong.rawValue), N := 1);
modbusLong.lowWord := OSCAT_BASIC.WORD_OF_DWORD(in := DINT_TO_DWORD(modbusLong.rawValue), N := 0);
END_METHOD

END_FUNCTION_BLOCK

// Device/Application/FBs/Motors/Applied Motion/Modbus Commands/FB_SendMoveCommandAppliedMotionTCP
FUNCTION_BLOCK FB_SendMoveCommandAppliedMotionTCP
VAR_INPUT
    distanceHighWord : WORD;
    distanceLowWord : WORD;        
    acceleration : INT;        //Acceleration in RPM/sec
    deceleration : INT;        //Deceleration in RPM/sec
    velocity : INT;            //Velocity in .25RPM
    opcode : STEP_SERVO_OPCODES;    //Opcode to perform
END_VAR
VAR_IN_OUT
    Slave :  IoDrvModbusTCP.ModbusTCPSlave;
END_VAR

VAR_OUTPUT
    xDone : BOOL;        //Successfully performed action
END_VAR
VAR
    moveCommandState : MOVE_MODBUS_COMMAND_STATES;
    modbusRequestTCP: IoDrvModbusTCP.ModbusRequest;
    modbusCommandTCP : IoDrvModbusTCP.ModbusCommand;
    sendBuffer : ARRAY [0 .. 4] OF WORD;            //Array of registers to send
    xExecute : BOOL;
    xExecuteONS : R_TRIG();
END_VAR

modbusRequestTCP(
                                slave:= Slave , 
                                xExecute:= , 
                                xAbort:= , 
                                usiUnitID:= , 
                                ModbusCommand:= modbusCommandTCP, 
                                pSendData:= ADR(sendBuffer), 
                                pRecvData:= , 
                                xBusy=> , 
                                xDone=> , 
                                xError=> , 
                                xAborted=> , 
                                ModbusError=> );

